   VAR
      ss_FB_HeartbeatPulse { ExternalAccessible := 'False'; ExternalVisible := 'False'; ExternalWritable := 'False'; S7_SetPoint := 'False'} : "FB_Pulse";   // Heartbeat send pulse generator
      s_UDT_MessageArray { ExternalAccessible := 'False'; ExternalVisible := 'False'; ExternalWritable := 'False'; S7_SetPoint := 'False'} : "UDT_MessageV2";   // Message array byte
      s_UDT_MessageHeader { ExternalAccessible := 'False'; ExternalVisible := 'False'; ExternalWritable := 'False'; S7_SetPoint := 'False'} : "UDT_MessageHeaderV2";   // Message header
      ss_Status { ExternalAccessible := 'False'; ExternalVisible := 'False'; ExternalWritable := 'False'} : Struct   // Status structure
         FIFOStatus { ExternalAccessible := 'False'; ExternalVisible := 'False'; ExternalWritable := 'False'} : "UDT_FifoStatus";
         FIFOError { ExternalAccessible := 'False'; ExternalVisible := 'False'; ExternalWritable := 'False'; S7_SetPoint := 'True'} : Bool;   //  FIFO error
         FIFOWarning { ExternalAccessible := 'False'; ExternalVisible := 'False'; ExternalWritable := 'False'; S7_SetPoint := 'True'} : Bool;   // FIFO warning
         InvalidMessageArraySize { ExternalAccessible := 'False'; ExternalVisible := 'False'; ExternalWritable := 'False'} : Bool;   // Message array is too short for message
         InvalidTimeInterval { ExternalAccessible := 'False'; ExternalVisible := 'False'; ExternalWritable := 'False'} : Bool;   // Heartbeat time interval lower than zero
      END_STRUCT;
      sdi_SerializePosition { ExternalAccessible := 'False'; ExternalVisible := 'False'; ExternalWritable := 'False'} : DInt;   // Position in array where serialize finished writing data +1
      si_MaximumMessageLength { ExternalAccessible := 'False'; ExternalVisible := 'False'; ExternalWritable := 'False'} : Int;   // Maximum number of elements in message array
      si_SerializeStatus { ExternalAccessible := 'False'; ExternalVisible := 'False'; ExternalWritable := 'False'} : Int;   // Function serialize status
      sx_HeartbeatPulse { ExternalAccessible := 'False'; ExternalVisible := 'False'; ExternalWritable := 'False'} : Bool;   // Heartbeat pulse
   END_VAR

   VAR CONSTANT
      ci_MessageID : Int := 20;   // Message ID number
      ci_MessageLength : Int := 18;   // Message length in bytes
   END_VAR


BEGIN
	(*
	----------------------------------------------------------------------------------------
	|                                                                                      |
	|  Copyright  2023             FORTNA Europe BV                                        |
	|  All Rights Reserved         Netherlands                                             |
	|                                                                                      |
	----------------------------------------------------------------------------------------
	Version history:
	Date        | Version   | Author       | Remark
	----------------------------------------------------------------------------------------
	03/01/2023  | 1.0       | S. Nikodem   | Release TIA 17 | DHL Munich 2023
	13/03/2023  | 1.1       | S. Nieswiec  | Updated for new Baseline
	*)
	REGION 1 – FIFO header status update

	    // Mode 'S' - FIFO register status update.
	    "FC_Fifo"(ic_Mode := 'S',
	              qUDT_Status => #ss_Status.FIFOStatus,
	              qx_Error => #ss_Status.FIFOError,
	              qx_Warning => #ss_Status.FIFOWarning,
	              iqv_Data := #s_UDT_MessageArray,
	              iqUDT_FifoHeader := #iq_UDT_FifoHeader,
	              iqv_DataBuffer := #iqs_FifoData);

	END_REGION

	REGION 2 – Heartbeat interval validation

	    // Check Heartbeat interval.
	    #ss_Status.InvalidTimeInterval := #iudi_HeartbeatInterval <= 0;

	END_REGION

	REGION 3 – Message array size validation

	    // Get size of the array.
	    #si_MaximumMessageLength := "FC_GetNrOfArrayEl"(#s_UDT_MessageArray.Bytes);

	    // Message array size validation.
	    #ss_Status.InvalidMessageArraySize := #ci_MessageLength > #si_MaximumMessageLength;

	END_REGION

	REGION 4 - Generate heartbeat pulse

	    IF NOT #ss_Status.InvalidTimeInterval
	        AND NOT #ss_Status.InvalidMessageArraySize
	    THEN
	        // Heartbeat pulse generator.
	        #ss_FB_HeartbeatPulse(iudi_PulseTime := #iudi_HeartbeatInterval,
	                              qx_Pulse => #sx_HeartbeatPulse);
	    END_IF;

	END_REGION

	REGION 5 – Message preparation

	    // FIFO full check.
	    IF NOT #iq_UDT_FifoHeader.Status.Full
	    THEN
	        // Errors and send pulse check.
	        IF NOT #ss_Status.FIFOError
	            AND NOT #ss_Status.InvalidMessageArraySize
	            AND #sx_HeartbeatPulse
	        THEN

	            REGION 5.1 – Header preparation

	                // Check sequence number. If it is equal or greater than 30000 reset it to 1.
	                IF #iqdi_MessageSequenceNumber < 30000
	                THEN
	                    #iqdi_MessageSequenceNumber += 1;
	                ELSE
	                    #iqdi_MessageSequenceNumber := 1;
	                END_IF;

	                // Write parts of the header into structure.
	                #s_UDT_MessageHeader.BodyLength := 0;
	                #s_UDT_MessageHeader.FlagRetry.%X0 := #ix_FlagRetry;
	                #s_UDT_MessageHeader.Group := #ii_MessageGroup;
	                #s_UDT_MessageHeader.MessageID := #ci_MessageID;
	                #s_UDT_MessageHeader.SequenceNumber := #iqdi_MessageSequenceNumber;
	                #s_UDT_MessageHeader.TimeSpan := #idi_TimeSpan;

	                // Calculate the header checksum.
	                "FC_Checksum"(i_UDT_MessageHeader := #s_UDT_MessageHeader,
	                              qb_Checksum => #s_UDT_MessageHeader.Checksum);

	            END_REGION

	            REGION 5.2 – Convert header into array of bytes

	                // Initialize the header serialize position and convert header structure into array of bytes.
	                #sdi_SerializePosition := 0;
	                #si_SerializeStatus := Serialize(SRC_VARIABLE := #s_UDT_MessageHeader,
	                                                 DEST_ARRAY => #s_UDT_MessageArray.Bytes,
	                                                 POS := #sdi_SerializePosition);

	            END_REGION

	            REGION 5.3 – Write message into the FIFO buffer

	                // Mode 'W' - Write FIFO record.
	                "FC_Fifo"(ic_Mode := 'W',
	                          qUDT_Status => #ss_Status.FIFOStatus,
	                          qx_Error => #ss_Status.FIFOError,
	                          qx_Warning => #ss_Status.FIFOWarning,
	                          iqv_Data := #s_UDT_MessageArray,
	                          iqUDT_FifoHeader := #iq_UDT_FifoHeader,
	                          iqv_DataBuffer := #iqs_FifoData);

	            END_REGION

	        END_IF;
	    ELSE
	        // If FIFO is full set FIFO main and FIFO full errors.
	        #ss_Status.FIFOError := TRUE;
	        #ss_Status.FIFOStatus.FifoFull := TRUE;
	    END_IF;

	END_REGION

	REGION 6 - Status

	    // Parametrization collective error output.
	    #qx_Error :=
	    #ss_Status.FIFOError
	    OR #ss_Status.InvalidTimeInterval
	    OR #ss_Status.InvalidMessageArraySize;

	    // Parametrization collective warning output.
	    #qx_Warning := #ss_Status.FIFOWarning;

	END_REGION
END_FUNCTION_BLOCK

FUNCTION_BLOCK "FB_MFC_Visu_PNNode_Status"
{ S7_Optimized_Access := 'TRUE' }
VERSION : 0.1
// ATTRIBUTES
// AUTO_NUMBER = True
// BLOCK_NUMBER = 155
// END_ATTRIBUTES
   VAR_INPUT
      i_UDT_PNNodeStatus { ExternalAccessible := 'False'; ExternalVisible := 'False'; ExternalWritable := 'False'} : "UDT_PNNodeStatus";   // PNNode status structure
      i_UDT_EquipmentNumber { ExternalAccessible := 'False'; ExternalVisible := 'False'; ExternalWritable := 'False'} : "UDT_EquipmentNumber";   // Item number
      ix_SendAllErrorsState { ExternalAccessible := 'False'; ExternalVisible := 'False'; ExternalWritable := 'False'} : Bool;   // True - update all the messages
      ix_MFCConnected { ExternalAccessible := 'False'; ExternalVisible := 'False'; ExternalWritable := 'False'} : Bool;   // True - A connection to the MFC has been established
      ix_CollectiveReset { ExternalAccessible := 'False'; ExternalVisible := 'False'; ExternalWritable := 'False'} : Bool;   // True - Collective reset command of all system controls
   END_VAR

   VAR_OUTPUT
      qx_Error { ExternalAccessible := 'False'; ExternalVisible := 'False'; ExternalWritable := 'False'} : Bool;   // Block error
      qx_Warning { ExternalAccessible := 'False'; ExternalVisible := 'False'; ExternalWritable := 'False'} : Bool;   // Block warning
   END_VAR

   VAR_IN_OUT
      iq_UDT_FifoHeader : "UDT_FifoHeader";   // FIFO header
      iqs_FifoData : Array[*] of "UDT_MessageV2";   // FIFO data buffer
      iqdi_MessageSequenceNumber { ExternalAccessible := 'False'; ExternalVisible := 'False'; ExternalWritable := 'False'} : DInt;   // Message number
   END_VAR

   VAR
      s_FB_ItemError { ExternalAccessible := 'False'; ExternalVisible := 'False'; ExternalWritable := 'False'; S7_SetPoint := 'False'} : "FB_ItemError";   // Item error block's instance
      s_FB_ItemStatus { ExternalAccessible := 'False'; ExternalVisible := 'False'; ExternalWritable := 'False'; S7_SetPoint := 'False'} : "FB_ItemStatus";   // Item status block's instance
      ss_FIFOStatus { ExternalAccessible := 'False'; ExternalVisible := 'False'; ExternalWritable := 'False'; S7_SetPoint := 'False'} : "UDT_FifoStatus";   // Status structure
      s_UDT_Message { ExternalAccessible := 'False'; ExternalVisible := 'False'; ExternalWritable := 'False'; S7_SetPoint := 'False'} : "UDT_MessageV2";   // Message
      s_UDT_PNNodeOld { ExternalAccessible := 'False'; ExternalVisible := 'False'; ExternalWritable := 'False'; S7_SetPoint := 'False'} : "UDT_PNNodeStatus";   // PNNode old status structure
      s_UDT_ItemError { ExternalAccessible := 'False'; ExternalVisible := 'False'; ExternalWritable := 'False'; S7_SetPoint := 'False'} : "UDT_ItemError";   // Item error message body structure
      s_UDT_ItemStatus { ExternalAccessible := 'False'; ExternalVisible := 'False'; ExternalWritable := 'False'; S7_SetPoint := 'False'} : "UDT_ItemStatus";   // Item status message body structure
      s_R_TRIG_Connection {InstructionName := 'R_TRIG'; LibVersion := '1.0'; ExternalAccessible := 'False'; ExternalVisible := 'False'; ExternalWritable := 'False'; S7_SetPoint := 'False'} : R_TRIG;   // Rising edge trigger connection reastablished
      s_F_TRIG_SendAllErrors {InstructionName := 'F_TRIG'; LibVersion := '1.0'; ExternalAccessible := 'False'; ExternalVisible := 'False'; ExternalWritable := 'False'; S7_SetPoint := 'False'} : F_TRIG;   // Falling edge trigger from signal send all errors
      sdi_Code { ExternalAccessible := 'False'; ExternalVisible := 'False'; ExternalWritable := 'False'} : DInt;   // Error code
      si_ItemStatus { ExternalAccessible := 'False'; ExternalVisible := 'False'; ExternalWritable := 'False'} : Int;   // Item status
      ii_ErrorNumber { ExternalAccessible := 'False'; ExternalVisible := 'False'; ExternalWritable := 'False'} : Int;   // Counter Error Number
      si_State { ExternalAccessible := 'False'; ExternalVisible := 'False'; ExternalWritable := 'False'} : Int;   // Error state
      sx_ItemErrorMessageReq { ExternalAccessible := 'False'; ExternalVisible := 'False'; ExternalWritable := 'False'} : Bool;   // Item error message required
      sx_ItemStatusMessageReq { ExternalAccessible := 'False'; ExternalVisible := 'False'; ExternalWritable := 'False'} : Bool;   // Item status message required
      sx_SendAllProcedure { ExternalAccessible := 'False'; ExternalVisible := 'False'; ExternalWritable := 'False'} : Bool;   // Send all procedure
      sx_FIFOError { ExternalAccessible := 'False'; ExternalVisible := 'False'; ExternalWritable := 'False'} : Bool;   // FIFO error
      sx_FIFOWarning { ExternalAccessible := 'False'; ExternalVisible := 'False'; ExternalWritable := 'False'} : Bool;   // FIFO warning
      sx_ItemErrorBlockError { ExternalAccessible := 'False'; ExternalVisible := 'False'; ExternalWritable := 'False'} : Bool;   // Item error block error
      sx_ItemErrorBlockWarning { ExternalAccessible := 'False'; ExternalVisible := 'False'; ExternalWritable := 'False'} : Bool;   // Item error block warning
      sx_ItemStatusBlockError { ExternalAccessible := 'False'; ExternalVisible := 'False'; ExternalWritable := 'False'} : Bool;   // Item status block error
      sx_ItemStatusBlockWarning { ExternalAccessible := 'False'; ExternalVisible := 'False'; ExternalWritable := 'False'} : Bool;   // Item status block warning
   END_VAR


BEGIN
	(*
	----------------------------------------------------------------------------------------
	|                                                                                      |
	|  Copyright  2023             FORTNA Europe BV                                        |
	|  All Rights Reserved         Netherlands                                             |
	|                                                                                      |
	----------------------------------------------------------------------------------------
	Version history:
	Date        | Version   | Author       | Remark
	----------------------------------------------------------------------------------------
	24/03/2023  | 1.0       | M. Diebel   | Release TIA 17 | DHL Munich 2023
	13/03/2023  | 1.1       | S. Nieswiec  | Updated for new Baseline
	*)


	REGION 1 - Initialize message required signals

	    #sx_ItemErrorMessageReq := FALSE;
	    #sx_ItemStatusMessageReq := FALSE;

	    // On connection reestablish send last remembered status and error state ( status only when it's diffrent then 0 )
	    #s_R_TRIG_Connection(CLK := #ix_MFCConnected);

	    IF #s_R_TRIG_Connection.Q AND #si_ItemStatus <> 0
	    THEN
	        #sx_ItemStatusMessageReq := TRUE;
	    END_IF;

	    IF #s_R_TRIG_Connection.Q
	    THEN
	        #sx_ItemErrorMessageReq := TRUE;
	    END_IF;

	    // Prepare trigger on the collective reset signal.
	    #s_F_TRIG_SendAllErrors(CLK := #ix_SendAllErrorsState);

	    // When collective reset will go down, start send every equipment errors.
	    IF #s_F_TRIG_SendAllErrors.Q AND NOT #sx_SendAllProcedure
	    THEN
	        #ii_ErrorNumber := 0;
	        #sx_SendAllProcedure := TRUE;
	    END_IF;

	END_REGION

	REGION 2 - FIFO header status update

	    // Mode 'S' - FIFO register status update.
	    "FC_Fifo"(ic_Mode := 'S',
	              qUDT_Status => #ss_FIFOStatus,
	              qx_Error => #sx_FIFOError,
	              qx_Warning => #sx_FIFOWarning,
	              iqv_Data := #s_UDT_Message,
	              iqUDT_FifoHeader := #iq_UDT_FifoHeader,
	              iqv_DataBuffer := #iqs_FifoData);

	END_REGION

	REGION 3 - Prepare message data

	    // When there is no reset errors command, update status and errors.
	    IF NOT #ix_CollectiveReset
	        AND NOT #ss_FIFOStatus.FifoPreFull
	    THEN
	        // Status
	        IF (#i_UDT_PNNodeStatus.Status <> #s_UDT_PNNodeOld.Status OR (#sx_SendAllProcedure AND #ii_ErrorNumber = 0))
	        THEN
	            #sx_ItemStatusMessageReq := TRUE;
	            #si_ItemStatus := #i_UDT_PNNodeStatus.Status;
	            #s_UDT_PNNodeOld.Status := #i_UDT_PNNodeStatus.Status;
	        END_IF;


	        // Check which specific status changed, prepare code, change state and write new status into the old one.
	        IF (#i_UDT_PNNodeStatus.Specific.PNSlaveNotOnline <> #s_UDT_PNNodeOld.Specific.PNSlaveNotOnline AND NOT #sx_SendAllProcedure)
	            OR (#sx_SendAllProcedure AND #ii_ErrorNumber = 0)
	        THEN
	            #sdi_Code := "DB_MFC_ErrorCode".PNNode.PNSlaveNotOnline;
	            #si_State := BOOL_TO_INT(#i_UDT_PNNodeStatus.Specific.PNSlaveNotOnline);
	            #s_UDT_PNNodeOld.Specific.PNSlaveNotOnline := #i_UDT_PNNodeStatus.Specific.PNSlaveNotOnline;
	            #sx_ItemErrorMessageReq := TRUE;
	            #ii_ErrorNumber += 1;
	        ELSIF (#i_UDT_PNNodeStatus.Specific.PNSlaveError <> #s_UDT_PNNodeOld.Specific.PNSlaveError AND NOT #sx_SendAllProcedure)
	            OR (#sx_SendAllProcedure AND #ii_ErrorNumber = 1)
	        THEN
	            #sdi_Code := "DB_MFC_ErrorCode".PNNode.PNSlaveError;
	            #si_State := BOOL_TO_INT(#i_UDT_PNNodeStatus.Specific.PNSlaveError);
	            #s_UDT_PNNodeOld.Specific.PNSlaveError := #i_UDT_PNNodeStatus.Specific.PNSlaveError;
	            #sx_ItemErrorMessageReq := TRUE;
	            #ii_ErrorNumber += 1;
	        ELSIF (#i_UDT_PNNodeStatus.Specific.PNSlaveWarning <> #s_UDT_PNNodeOld.Specific.PNSlaveWarning AND NOT #sx_SendAllProcedure)
	            OR (#sx_SendAllProcedure AND #ii_ErrorNumber = 2)
	        THEN
	            #sdi_Code := "DB_MFC_ErrorCode".PNNode.PNSlaveWarning;
	            #si_State := BOOL_TO_INT(#i_UDT_PNNodeStatus.Specific.PNSlaveWarning);
	            #s_UDT_PNNodeOld.Specific.PNSlaveWarning := #i_UDT_PNNodeStatus.Specific.PNSlaveWarning;
	            #sx_ItemErrorMessageReq := TRUE;
	            #sx_SendAllProcedure := FALSE;
	            #ii_ErrorNumber += 1;
	        END_IF;
	    END_IF;
	END_REGION

	REGION 4 - Write message components to the item error structure

	    #s_UDT_ItemError.ItemNumber := #i_UDT_EquipmentNumber;
	    #s_UDT_ItemError.Error := #sdi_Code;
	    #s_UDT_ItemError.State := #si_State;
	    #s_UDT_ItemError.Masked := 1;

	END_REGION

	REGION 5 - Write message components to the item status structure

	    #s_UDT_ItemStatus.Group := #i_UDT_EquipmentNumber.Group;
	    #s_UDT_ItemStatus.Node := #i_UDT_EquipmentNumber.Node;
	    #s_UDT_ItemStatus.Status := #si_ItemStatus;

	END_REGION

	REGION 6 - Prepare messages to the MFC

	    // If item error message required signal is set, prepare the item error message.
	    IF (#sx_ItemErrorMessageReq)
	    THEN
	        #s_FB_ItemError(i_UDT_ItemErrorBody := #s_UDT_ItemError,
	                        ii_MessageGroup := 1,
	                        ix_FlagRetry := FALSE,
	                        idi_TimeSpan := 0,
	                        qx_Error => #sx_ItemErrorBlockError,
	                        qx_Warning => #sx_ItemErrorBlockWarning,
	                        iq_UDT_FifoHeader := #iq_UDT_FifoHeader,
	                        iqs_FifoData := #iqs_FifoData,
	                        iqdi_MessageSequenceNumber := #iqdi_MessageSequenceNumber);
	    END_IF;

	    // If item status message required signal is set, prepare the item error message.
	    IF (#sx_ItemStatusMessageReq)
	    THEN
	        #s_FB_ItemStatus(i_UDT_ItemStatusBody := #s_UDT_ItemStatus,
	                         ii_MessageGroup := 1,
	                         ix_FlagRetry := FALSE,
	                         idi_TimeSpan := 0,
	                         qx_Error => #sx_ItemStatusBlockError,
	                         qx_Warning => #sx_ItemStatusBlockWarning,
	                         iq_UDT_FifoHeader := #iq_UDT_FifoHeader,
	                         iqs_FifoData := #iqs_FifoData,
	                         iqdi_MessageSequenceNumber := #iqdi_MessageSequenceNumber);
	    END_IF;

	END_REGION

	REGION 7 - Write outputs

	    // Prepare collective output error.
	    #qx_Error :=
	    #sx_ItemErrorBlockError
	    OR #sx_ItemStatusBlockError
	    OR #sx_FIFOError;

	    // Prepare collective output warning.
	    #qx_Warning :=
	    #sx_ItemErrorBlockWarning
	    OR #sx_ItemStatusBlockWarning
	    OR #sx_FIFOWarning;

	END_REGION
END_FUNCTION_BLOCK

FUNCTION_BLOCK "FB_MFC_Visu_EuchnerLock"
{ S7_Optimized_Access := 'TRUE' }
VERSION : 0.1
// ATTRIBUTES
// AUTO_NUMBER = True
// BLOCK_NUMBER = 149
// END_ATTRIBUTES
   VAR_INPUT
      i_UDT_EuchnerLock { ExternalAccessible := 'False'; ExternalVisible := 'False'; ExternalWritable := 'False'} : "UDT_EuchnerLockStatusV2";
      i_UDT_EquipmentNumber { ExternalAccessible := 'False'; ExternalVisible := 'False'; ExternalWritable := 'False'} : "UDT_EquipmentNumber";   // Item number
      ix_SendAllErrorsState { ExternalAccessible := 'False'; ExternalVisible := 'False'; ExternalWritable := 'False'} : Bool;   // True - update all the messages
      ix_MFCConnected { ExternalAccessible := 'False'; ExternalVisible := 'False'; ExternalWritable := 'False'} : Bool;   // True - A connection to the MFC has been established
      ix_CollectiveReset { ExternalAccessible := 'False'; ExternalVisible := 'False'; ExternalWritable := 'False'} : Bool;   // True - Collective reset command of all system controls
   END_VAR

   VAR_OUTPUT
      qx_Error { ExternalAccessible := 'False'; ExternalVisible := 'False'; ExternalWritable := 'False'} : Bool;   // Block error
      qx_Warning { ExternalAccessible := 'False'; ExternalVisible := 'False'; ExternalWritable := 'False'} : Bool;   // Block warning
   END_VAR

   VAR_IN_OUT
      iq_UDT_FifoHeader : "UDT_FifoHeader";   // FIFO header
      iqs_FifoData : Array[*] of "UDT_MessageV2";   // FIFO data buffer
      iqdi_MessageSequenceNumber { ExternalAccessible := 'False'; ExternalVisible := 'False'; ExternalWritable := 'False'} : DInt;   // Message number
   END_VAR

   VAR
      s_FB_ItemError { ExternalAccessible := 'False'; ExternalVisible := 'False'; ExternalWritable := 'False'; S7_SetPoint := 'False'} : "FB_ItemError";   // Item error block's instance
      s_FB_ItemStatus { ExternalAccessible := 'False'; ExternalVisible := 'False'; ExternalWritable := 'False'; S7_SetPoint := 'False'} : "FB_ItemStatus";   // Item status block's instance
      ss_FIFOStatus { ExternalAccessible := 'False'; ExternalVisible := 'False'; ExternalWritable := 'False'; S7_SetPoint := 'False'} : "UDT_FifoStatus";   // Status structure
      s_UDT_Message { ExternalAccessible := 'False'; ExternalVisible := 'False'; ExternalWritable := 'False'; S7_SetPoint := 'False'} : "UDT_MessageV2";   // Message
      s_UDT_EuchnerLockOld { ExternalAccessible := 'False'; ExternalVisible := 'False'; ExternalWritable := 'False'; S7_SetPoint := 'False'} : "UDT_EuchnerLockStatusV2";   // ColumnLift status structure
      s_UDT_ItemError { ExternalAccessible := 'False'; ExternalVisible := 'False'; ExternalWritable := 'False'; S7_SetPoint := 'False'} : "UDT_ItemError";   // Item error message body structure
      s_UDT_ItemStatus { ExternalAccessible := 'False'; ExternalVisible := 'False'; ExternalWritable := 'False'; S7_SetPoint := 'False'} : "UDT_ItemStatus";   // Item status message body structure
      s_R_TRIG_Connection {InstructionName := 'R_TRIG'; LibVersion := '1.0'; ExternalAccessible := 'False'; ExternalVisible := 'False'; ExternalWritable := 'False'; S7_SetPoint := 'False'} : R_TRIG;   // Rising edge trigger connection reastablished
      s_F_TRIG_SendAllErrors {InstructionName := 'F_TRIG'; LibVersion := '1.0'; ExternalAccessible := 'False'; ExternalVisible := 'False'; ExternalWritable := 'False'; S7_SetPoint := 'False'} : F_TRIG;   // Falling edge trigger from signal send all errors
      sdi_Code { ExternalAccessible := 'False'; ExternalVisible := 'False'; ExternalWritable := 'False'} : DInt;   // Error code
      si_ItemStatus { ExternalAccessible := 'False'; ExternalVisible := 'False'; ExternalWritable := 'False'} : Int;   // Item status
      ii_ErrorNumber { ExternalAccessible := 'False'; ExternalVisible := 'False'; ExternalWritable := 'False'} : Int;   // Counter Error Number
      si_State { ExternalAccessible := 'False'; ExternalVisible := 'False'; ExternalWritable := 'False'} : Int;   // Error state
      sx_ItemErrorMessageReq { ExternalAccessible := 'False'; ExternalVisible := 'False'; ExternalWritable := 'False'} : Bool;   // Item error message required
      sx_ItemStatusMessageReq { ExternalAccessible := 'False'; ExternalVisible := 'False'; ExternalWritable := 'False'} : Bool;   // Item status message required
      sx_SendAllProcedure { ExternalAccessible := 'False'; ExternalVisible := 'False'; ExternalWritable := 'False'} : Bool;   // Send all procedure
      sx_FIFOError { ExternalAccessible := 'False'; ExternalVisible := 'False'; ExternalWritable := 'False'} : Bool;   // FIFO error
      sx_FIFOWarning { ExternalAccessible := 'False'; ExternalVisible := 'False'; ExternalWritable := 'False'} : Bool;   // FIFO warning
      sx_ItemErrorBlockError { ExternalAccessible := 'False'; ExternalVisible := 'False'; ExternalWritable := 'False'} : Bool;   // Item error block error
      sx_ItemErrorBlockWarning { ExternalAccessible := 'False'; ExternalVisible := 'False'; ExternalWritable := 'False'} : Bool;   // Item error block warning
      sx_ItemStatusBlockError { ExternalAccessible := 'False'; ExternalVisible := 'False'; ExternalWritable := 'False'} : Bool;   // Item status block error
      sx_ItemStatusBlockWarning { ExternalAccessible := 'False'; ExternalVisible := 'False'; ExternalWritable := 'False'} : Bool;   // Item status block warning
      s_UDT_EuchnerLockStatus { ExternalAccessible := 'False'; ExternalVisible := 'False'; ExternalWritable := 'False'; S7_SetPoint := 'False'} : "UDT_EuchnerLockStatusV2";   // ColumnLift status structure
   END_VAR


BEGIN
	(*
	----------------------------------------------------------------------------------------
	|                                                                                      |
	|  Copyright  2023             FORTNA Europe BV                                        |
	|  All Rights Reserved         Netherlands                                             |
	|                                                                                      |
	----------------------------------------------------------------------------------------
	Version history:
	Date        | Version   | Author       | Remark
	----------------------------------------------------------------------------------------
	10/10/2023  | 1.0       | M. Diebel   | Release TIA 17 | DHL Munich 2023
	06/02/2024  | 1.1       | L.Klar      | New alarms added
	13/03/2023  | 1.2       | S. Nieswiec  | Updated for new Baseline
	*)


	REGION 1 - Initialize message required signals


	    #sx_ItemErrorMessageReq := FALSE;
	    #sx_ItemStatusMessageReq := FALSE;

	    // On connection reestablish send last remembered status and error state ( status only when it's diffrent then 0 )
	    #s_R_TRIG_Connection(CLK := #ix_MFCConnected);

	    IF #s_R_TRIG_Connection.Q AND #si_ItemStatus <> 0
	    THEN
	        #sx_ItemStatusMessageReq := TRUE;
	    END_IF;

	    IF #s_R_TRIG_Connection.Q
	    THEN
	        #sx_ItemErrorMessageReq := TRUE;
	    END_IF;

	    // Prepare trigger on the collective reset signal.
	    #s_F_TRIG_SendAllErrors(CLK := #ix_SendAllErrorsState);

	    // When collective reset will go down, start send every equipment errors.
	    IF #s_F_TRIG_SendAllErrors.Q AND NOT #sx_SendAllProcedure
	    THEN
	        #ii_ErrorNumber := 0;
	        #sx_SendAllProcedure := TRUE;
	    END_IF;

	END_REGION

	REGION 2 - FIFO header status update

	    // Mode 'S' - FIFO register status update.
	    "FC_Fifo"(ic_Mode := 'S',
	              qUDT_Status => #ss_FIFOStatus,
	              qx_Error => #sx_FIFOError,
	              qx_Warning => #sx_FIFOWarning,
	              iqv_Data := #s_UDT_Message,
	              iqUDT_FifoHeader := #iq_UDT_FifoHeader,
	              iqv_DataBuffer := #iqs_FifoData);

	END_REGION

	REGION 3 - Prepare message data

	    //
	    #s_UDT_EuchnerLockStatus := #i_UDT_EuchnerLock;
	    // When there is no reset errors command, update status and errors.
	    IF NOT #ix_CollectiveReset
	        AND NOT #ss_FIFOStatus.FifoPreFull
	    THEN


	        // Check which specific status changed, prepare code, change state and write new status into the old one.
	        IF (#s_UDT_EuchnerLockStatus.LockFault <> #s_UDT_EuchnerLockOld.LockFault AND NOT #sx_SendAllProcedure)
	            OR (#sx_SendAllProcedure AND #ii_ErrorNumber = 0)
	        THEN
	            #sdi_Code := "DB_MFC_ErrorCode".EuchnerLock.LockFault;
	            #si_State := BOOL_TO_INT(#s_UDT_EuchnerLockStatus.LockFault);
	            #s_UDT_EuchnerLockOld.LockFault := #s_UDT_EuchnerLockStatus.LockFault;
	            #sx_ItemErrorMessageReq := TRUE;
	            #ii_ErrorNumber += 1;
	        ELSIF (#s_UDT_EuchnerLockStatus.DoorClosed <> #s_UDT_EuchnerLockOld.DoorClosed AND NOT #sx_SendAllProcedure)
	            OR (#sx_SendAllProcedure AND #ii_ErrorNumber = 1)
	        THEN
	            #sdi_Code := "DB_MFC_ErrorCode".EuchnerLock.DoorClosed;
	            #si_State := BOOL_TO_INT(#s_UDT_EuchnerLockStatus.DoorClosed);
	            #s_UDT_EuchnerLockOld.DoorClosed := #s_UDT_EuchnerLockStatus.DoorClosed;
	            #sx_ItemErrorMessageReq := TRUE;
	            #ii_ErrorNumber += 1;
	        ELSIF (#s_UDT_EuchnerLockStatus.DoorOpened <> #s_UDT_EuchnerLockOld.DoorOpened AND NOT #sx_SendAllProcedure)
	            OR (#sx_SendAllProcedure AND #ii_ErrorNumber = 2)
	        THEN
	            #sdi_Code := "DB_MFC_ErrorCode".EuchnerLock.DoorOpened;
	            #si_State := BOOL_TO_INT(#s_UDT_EuchnerLockStatus.DoorOpened);
	            #s_UDT_EuchnerLockOld.DoorOpened := #s_UDT_EuchnerLockStatus.DoorOpened;
	            #sx_ItemErrorMessageReq := TRUE;
	            #ii_ErrorNumber += 1;
	        ELSIF (#s_UDT_EuchnerLockStatus.BoltTongueClosed <> #s_UDT_EuchnerLockOld.BoltTongueClosed AND NOT #sx_SendAllProcedure)
	            OR (#sx_SendAllProcedure AND #ii_ErrorNumber = 3)
	        THEN
	            #sdi_Code := "DB_MFC_ErrorCode".EuchnerLock.BoltTongueClosed;
	            #si_State := BOOL_TO_INT(#s_UDT_EuchnerLockStatus.BoltTongueClosed);
	            #s_UDT_EuchnerLockOld.BoltTongueClosed := #s_UDT_EuchnerLockStatus.BoltTongueClosed;
	            #sx_ItemErrorMessageReq := TRUE;
	            #ii_ErrorNumber += 1;
	        ELSIF (#s_UDT_EuchnerLockStatus.Safelylocked <> #s_UDT_EuchnerLockOld.Safelylocked AND NOT #sx_SendAllProcedure)
	            OR (#sx_SendAllProcedure AND #ii_ErrorNumber = 4)
	        THEN
	            #sdi_Code := "DB_MFC_ErrorCode".EuchnerLock.Safelylocked;
	            #si_State := BOOL_TO_INT(#s_UDT_EuchnerLockStatus.Safelylocked);
	            #s_UDT_EuchnerLockOld.Safelylocked := #s_UDT_EuchnerLockStatus.Safelylocked;
	            #sx_ItemErrorMessageReq := TRUE;
	            #ii_ErrorNumber += 1;
	        ELSIF (#s_UDT_EuchnerLockStatus.SafetyLockAckReq <> #s_UDT_EuchnerLockOld.SafetyLockAckReq AND NOT #sx_SendAllProcedure)
	            OR (#sx_SendAllProcedure AND #ii_ErrorNumber = 5)
	        THEN
	            #sdi_Code := "DB_MFC_ErrorCode".EuchnerLock.SafetyLockAckReq;
	            #si_State := BOOL_TO_INT(#s_UDT_EuchnerLockStatus.SafetyLockAckReq);
	            #s_UDT_EuchnerLockOld.SafetyLockAckReq := #s_UDT_EuchnerLockStatus.SafetyLockAckReq;
	            #sx_ItemErrorMessageReq := TRUE;
	            #ii_ErrorNumber += 1;
	        ELSIF (#s_UDT_EuchnerLockStatus.ReqMissingAccessRights <> #s_UDT_EuchnerLockOld.ReqMissingAccessRights AND NOT #sx_SendAllProcedure)
	            OR (#sx_SendAllProcedure AND #ii_ErrorNumber = 6)
	        THEN
	            #sdi_Code := "DB_MFC_ErrorCode".EuchnerLock.ReqMissingAccessRights;
	            #si_State := BOOL_TO_INT(#s_UDT_EuchnerLockStatus.ReqMissingAccessRights);
	            #s_UDT_EuchnerLockOld.ReqMissingAccessRights := #s_UDT_EuchnerLockStatus.ReqMissingAccessRights;
	            #sx_ItemErrorMessageReq := TRUE;
	            #ii_ErrorNumber += 1;
	        ELSIF (#s_UDT_EuchnerLockStatus.ResetMissingAccessRights <> #s_UDT_EuchnerLockOld.ResetMissingAccessRights AND NOT #sx_SendAllProcedure)
	            OR (#sx_SendAllProcedure AND #ii_ErrorNumber = 7)
	        THEN
	            #sdi_Code := "DB_MFC_ErrorCode".EuchnerLock.ResetMissingAccessRights;
	            #si_State := BOOL_TO_INT(#s_UDT_EuchnerLockStatus.ResetMissingAccessRights);
	            #s_UDT_EuchnerLockOld.ResetMissingAccessRights := #s_UDT_EuchnerLockStatus.ResetMissingAccessRights;
	            #sx_ItemErrorMessageReq := TRUE;
	            #ii_ErrorNumber += 1;
	        ELSIF (#s_UDT_EuchnerLockStatus.DoorOpenedWithoutReq <> #s_UDT_EuchnerLockOld.DoorOpenedWithoutReq AND NOT #sx_SendAllProcedure)
	            OR (#sx_SendAllProcedure AND #ii_ErrorNumber = 8)
	        THEN
	            #sdi_Code := "DB_MFC_ErrorCode".EuchnerLock.DoorOpenedWithoutReq;
	            #si_State := BOOL_TO_INT(#s_UDT_EuchnerLockStatus.DoorOpenedWithoutReq);
	            #s_UDT_EuchnerLockOld.DoorOpenedWithoutReq := #s_UDT_EuchnerLockStatus.DoorOpenedWithoutReq;
	            #sx_ItemErrorMessageReq := TRUE;
	            #ii_ErrorNumber += 1;
	            #sx_SendAllProcedure := FALSE;
	        END_IF;
	    END_IF;
	END_REGION

	REGION 4 - Write message components to the item error structure

	    #s_UDT_ItemError.ItemNumber := #i_UDT_EquipmentNumber;
	    #s_UDT_ItemError.Error := #sdi_Code;
	    #s_UDT_ItemError.State := #si_State;
	    #s_UDT_ItemError.Masked := 1;

	END_REGION

	REGION 5 - Write message components to the item status structure

	    #s_UDT_ItemStatus.Group := #i_UDT_EquipmentNumber.Group;
	    #s_UDT_ItemStatus.Node := #i_UDT_EquipmentNumber.Node;
	    #s_UDT_ItemStatus.Status := #si_ItemStatus;

	END_REGION

	REGION 6 - Prepare messages to the MFC

	    // If item error message required signal is set, prepare the item error message.
	    IF (#sx_ItemErrorMessageReq)
	    THEN
	        #s_FB_ItemError(i_UDT_ItemErrorBody := #s_UDT_ItemError,
	                        ii_MessageGroup := 1,
	                        ix_FlagRetry := FALSE,
	                        idi_TimeSpan := 0,
	                        qx_Error => #sx_ItemErrorBlockError,
	                        qx_Warning => #sx_ItemErrorBlockWarning,
	                        iq_UDT_FifoHeader := #iq_UDT_FifoHeader,
	                        iqs_FifoData := #iqs_FifoData,
	                        iqdi_MessageSequenceNumber := #iqdi_MessageSequenceNumber);
	    END_IF;

	    // If item status message required signal is set, prepare the item error message.
	    IF (#sx_ItemStatusMessageReq)
	    THEN
	        #s_FB_ItemStatus(i_UDT_ItemStatusBody := #s_UDT_ItemStatus,
	                         ii_MessageGroup := 1,
	                         ix_FlagRetry := FALSE,
	                         idi_TimeSpan := 0,
	                         qx_Error => #sx_ItemStatusBlockError,
	                         qx_Warning => #sx_ItemStatusBlockWarning,
	                         iq_UDT_FifoHeader := #iq_UDT_FifoHeader,
	                         iqs_FifoData := #iqs_FifoData,
	                         iqdi_MessageSequenceNumber := #iqdi_MessageSequenceNumber);
	    END_IF;

	END_REGION

	REGION 7 - Write outputs

	    // Prepare collective output error.
	    #qx_Error :=
	    #sx_ItemErrorBlockError
	    OR #sx_ItemStatusBlockError
	    OR #sx_FIFOError;

	    // Prepare collective output warning.
	    #qx_Warning :=
	    #sx_ItemErrorBlockWarning
	    OR #sx_ItemStatusBlockWarning
	    OR #sx_FIFOWarning;

	END_REGION
END_FUNCTION_BLOCK

FUNCTION_BLOCK "FB_MFC_Visu_EStop_Status"
{ S7_Optimized_Access := 'TRUE' }
VERSION : 0.1
// ATTRIBUTES
// AUTO_NUMBER = True
// BLOCK_NUMBER = 148
// END_ATTRIBUTES
   VAR_INPUT
      i_UDT_EStopStatus { ExternalAccessible := 'False'; ExternalVisible := 'False'; ExternalWritable := 'False'} : "UDT_EStop_Status";   // EStop status structure
      i_UDT_EquipmentNumber { ExternalAccessible := 'False'; ExternalVisible := 'False'; ExternalWritable := 'False'} : "UDT_EquipmentNumber";   // Item number
      ix_SendAllErrorsState { ExternalAccessible := 'False'; ExternalVisible := 'False'; ExternalWritable := 'False'} : Bool;   // True - update all the messages
      ix_MFCConnected { ExternalAccessible := 'False'; ExternalVisible := 'False'; ExternalWritable := 'False'} : Bool;   // True - A connection to the MFC has been established
      ix_CollectiveReset { ExternalAccessible := 'False'; ExternalVisible := 'False'; ExternalWritable := 'False'} : Bool;   // True - Collective reset command of all system controls
   END_VAR

   VAR_OUTPUT
      qx_Error { ExternalAccessible := 'False'; ExternalVisible := 'False'; ExternalWritable := 'False'} : Bool;   // Block error
      qx_Warning { ExternalAccessible := 'False'; ExternalVisible := 'False'; ExternalWritable := 'False'} : Bool;   // Block warning
   END_VAR

   VAR_IN_OUT
      iq_UDT_FifoHeader : "UDT_FifoHeader";   // FIFO header
      iqs_FifoData : Array[*] of "UDT_MessageV2";   // FIFO data buffer
      iqdi_MessageSequenceNumber { ExternalAccessible := 'False'; ExternalVisible := 'False'; ExternalWritable := 'False'} : DInt;   // Message number
   END_VAR

   VAR
      s_FB_ItemStatus { ExternalAccessible := 'False'; ExternalVisible := 'False'; ExternalWritable := 'False'; S7_SetPoint := 'False'} : "FB_ItemStatus";   // Item status block's instance
      s_FB_ItemError { ExternalAccessible := 'False'; ExternalVisible := 'False'; ExternalWritable := 'False'; S7_SetPoint := 'False'} : "FB_ItemError";   // Item error block's instance
      ss_FIFOStatus { ExternalAccessible := 'False'; ExternalVisible := 'False'; ExternalWritable := 'False'; S7_SetPoint := 'False'} : "UDT_FifoStatus";   // Status structure
      s_UDT_Message { ExternalAccessible := 'False'; ExternalVisible := 'False'; ExternalWritable := 'False'; S7_SetPoint := 'False'} : "UDT_MessageV2";   // Message
      s_UDT_EStopOld { ExternalAccessible := 'False'; ExternalVisible := 'False'; ExternalWritable := 'False'; S7_SetPoint := 'False'} : "UDT_EStop_Status";   // EStop  status structure
      s_UDT_ItemError { ExternalAccessible := 'False'; ExternalVisible := 'False'; ExternalWritable := 'False'; S7_SetPoint := 'False'} : "UDT_ItemError";   // Item error message body structure
      s_UDT_ItemStatus { ExternalAccessible := 'False'; ExternalVisible := 'False'; ExternalWritable := 'False'; S7_SetPoint := 'False'} : "UDT_ItemStatus";   // Item status message body structure
      s_F_TRIG_SendAllErrors {InstructionName := 'F_TRIG'; LibVersion := '1.0'; ExternalAccessible := 'False'; ExternalVisible := 'False'; ExternalWritable := 'False'; S7_SetPoint := 'False'} : F_TRIG;   // Falling edge trigger from signal send all errors
      s_R_TRIG_Connection {InstructionName := 'R_TRIG'; LibVersion := '1.0'; ExternalAccessible := 'False'; ExternalVisible := 'False'; ExternalWritable := 'False'; S7_SetPoint := 'False'} : R_TRIG;   // Rising edge trigger connection reastablished
      sdi_Code { ExternalAccessible := 'False'; ExternalVisible := 'False'; ExternalWritable := 'False'} : DInt;   // Error code
      si_ItemStatus { ExternalAccessible := 'False'; ExternalVisible := 'False'; ExternalWritable := 'False'} : Int;   // Item status
      ii_ErrorNumber { ExternalAccessible := 'False'; ExternalVisible := 'False'; ExternalWritable := 'False'} : Int;   // Counter Error Number
      si_State { ExternalAccessible := 'False'; ExternalVisible := 'False'; ExternalWritable := 'False'} : Int;   // Error state
      sx_ItemErrorMessageReq { ExternalAccessible := 'False'; ExternalVisible := 'False'; ExternalWritable := 'False'} : Bool;   // Item error message required
      sx_ItemStatusMessageReq { ExternalAccessible := 'False'; ExternalVisible := 'False'; ExternalWritable := 'False'} : Bool;   // Item status message required
      sx_SendAllProcedure { ExternalAccessible := 'False'; ExternalVisible := 'False'; ExternalWritable := 'False'} : Bool;   // Send all procedure
      sx_FIFOError { ExternalAccessible := 'False'; ExternalVisible := 'False'; ExternalWritable := 'False'} : Bool;   // FIFO error
      sx_FIFOWarning { ExternalAccessible := 'False'; ExternalVisible := 'False'; ExternalWritable := 'False'} : Bool;   // FIFO warning
      sx_ItemErrorBlockError { ExternalAccessible := 'False'; ExternalVisible := 'False'; ExternalWritable := 'False'} : Bool;   // Item error block error
      sx_ItemErrorBlockWarning { ExternalAccessible := 'False'; ExternalVisible := 'False'; ExternalWritable := 'False'} : Bool;   // Item error block warning
      sx_ItemStatusBlockError { ExternalAccessible := 'False'; ExternalVisible := 'False'; ExternalWritable := 'False'} : Bool;   // Item status block error
      sx_ItemStatusBlockWarning { ExternalAccessible := 'False'; ExternalVisible := 'False'; ExternalWritable := 'False'} : Bool;   // Item status block warning
   END_VAR


BEGIN
	(*
	----------------------------------------------------------------------------------------
	|                                                                                      |
	|  Copyright  2023             FORTNA Europe BV                                        |
	|  All Rights Reserved         Netherlands                                             |
	|                                                                                      |
	----------------------------------------------------------------------------------------
	Version history:
	Date        | Version   | Author       | Remark
	----------------------------------------------------------------------------------------
	21/03/2023  | 1.0       | M. Diebel   | Release TIA 17 | DHL Munich 2023
	13/03/2023  | 1.1       | S. Nieswiec  | Updated for new Baseline
	*)


	REGION 1 - Initialize message required signals

	    #sx_ItemErrorMessageReq := FALSE;
	    #sx_ItemStatusMessageReq := FALSE;

	    // On connection reestablish send last remembered status and error state ( status only when it's diffrent then 0 )
	    #s_R_TRIG_Connection(CLK := #ix_MFCConnected);

	    IF #s_R_TRIG_Connection.Q AND #si_ItemStatus <> 0
	    THEN
	        #sx_ItemStatusMessageReq := TRUE;
	    END_IF;

	    IF #s_R_TRIG_Connection.Q
	    THEN
	        #sx_ItemErrorMessageReq := TRUE;
	    END_IF;

	    // Prepare trigger on the collective reset signal.
	    #s_F_TRIG_SendAllErrors(CLK := #ix_SendAllErrorsState);

	    // When collective reset will go down, start send every equipment errors.
	    IF #s_F_TRIG_SendAllErrors.Q AND NOT #sx_SendAllProcedure
	    THEN
	        #sx_SendAllProcedure := TRUE;
	    END_IF;

	END_REGION

	REGION 2 - FIFO header status update

	    // Mode 'S' - FIFO register status update.
	    "FC_Fifo"(ic_Mode := 'S',
	              qUDT_Status => #ss_FIFOStatus,
	              qx_Error => #sx_FIFOError,
	              qx_Warning => #sx_FIFOWarning,
	              iqv_Data := #s_UDT_Message,
	              iqUDT_FifoHeader := #iq_UDT_FifoHeader,
	              iqv_DataBuffer := #iqs_FifoData);

	END_REGION

	REGION 3 - Prepare message data

	    // When there is no reset errors command, update status and errors.
	    IF NOT #ix_CollectiveReset
	        AND NOT #ss_FIFOStatus.FifoPreFull
	    THEN
	        // Status
	        IF (#i_UDT_EStopStatus.Status <> #s_UDT_EStopOld.Status OR (#sx_SendAllProcedure))
	        THEN
	            #sx_ItemStatusMessageReq := TRUE;
	            #si_ItemStatus := #i_UDT_EStopStatus.Status;
	            #s_UDT_EStopOld.Status := #i_UDT_EStopStatus.Status;
	        END_IF;


	        // Check which specific status changed, prepare code, change state and write new status into the old one.
	        IF (#i_UDT_EStopStatus.Estop <> #s_UDT_EStopOld.Estop AND NOT #sx_SendAllProcedure)
	            OR (#sx_SendAllProcedure)
	        THEN
	            #sdi_Code := "DB_MFC_ErrorCode".EStop.EStop;
	            #si_State := BOOL_TO_INT(#i_UDT_EStopStatus.Estop);
	            #s_UDT_EStopOld.Estop := #i_UDT_EStopStatus.Estop;
	            #sx_ItemErrorMessageReq := TRUE;
	            #sx_SendAllProcedure := FALSE;
	        END_IF;
	    END_IF;
	END_REGION

	REGION 4 - Write message components to the item error structure

	    #s_UDT_ItemError.ItemNumber := #i_UDT_EquipmentNumber;
	    #s_UDT_ItemError.Error := #sdi_Code;
	    #s_UDT_ItemError.State := #si_State;
	    #s_UDT_ItemError.Masked := 1;

	END_REGION

	REGION 5 - Write message components to the item status structure

	    #s_UDT_ItemStatus.Group := #i_UDT_EquipmentNumber.Group;
	    #s_UDT_ItemStatus.Node := #i_UDT_EquipmentNumber.Node;
	    #s_UDT_ItemStatus.Status := #si_ItemStatus;

	END_REGION

	REGION 6 - Prepare messages to the MFC

	    // If item error message required signal is set, prepare the item error message.
	    IF (#sx_ItemErrorMessageReq)
	    THEN
	        #s_FB_ItemError(i_UDT_ItemErrorBody := #s_UDT_ItemError,
	                        ii_MessageGroup := 1,
	                        ix_FlagRetry := FALSE,
	                        idi_TimeSpan := 0,
	                        qx_Error => #sx_ItemErrorBlockError,
	                        qx_Warning => #sx_ItemErrorBlockWarning,
	                        iq_UDT_FifoHeader := #iq_UDT_FifoHeader,
	                        iqs_FifoData := #iqs_FifoData,
	                        iqdi_MessageSequenceNumber := #iqdi_MessageSequenceNumber);
	    END_IF;

	    // If item status message required signal is set, prepare the item error message.
	    IF (#sx_ItemStatusMessageReq)
	    THEN
	        #s_FB_ItemStatus(i_UDT_ItemStatusBody := #s_UDT_ItemStatus,
	                         ii_MessageGroup := 1,
	                         ix_FlagRetry := FALSE,
	                         idi_TimeSpan := 0,
	                         qx_Error => #sx_ItemStatusBlockError,
	                         qx_Warning => #sx_ItemStatusBlockWarning,
	                         iq_UDT_FifoHeader := #iq_UDT_FifoHeader,
	                         iqs_FifoData := #iqs_FifoData,
	                         iqdi_MessageSequenceNumber := #iqdi_MessageSequenceNumber);
	    END_IF;

	END_REGION

	REGION 7 - Write outputs

	    // Prepare collective output error.
	    #qx_Error :=
	    #sx_ItemErrorBlockError
	    OR #sx_ItemStatusBlockError
	    OR #sx_FIFOError;

	    // Prepare collective output warning.
	    #qx_Warning :=
	    #sx_ItemErrorBlockWarning
	    OR #sx_ItemStatusBlockWarning
	    OR #sx_FIFOWarning;

	END_REGION
END_FUNCTION_BLOCK

FUNCTION_BLOCK "FB_MFC_Visu_CPG_Status"
{ S7_Optimized_Access := 'TRUE' }
VERSION : 0.1
// ATTRIBUTES
// AUTO_NUMBER = True
// BLOCK_NUMBER = 142
// END_ATTRIBUTES
   VAR_INPUT
      i_UDT_CPGStatus { ExternalAccessible := 'False'; ExternalVisible := 'False'; ExternalWritable := 'False'} : "UDT_ControlPowerGroupWORStatus";   // CPG status structure
      i_UDT_EquipmentNumber { ExternalAccessible := 'False'; ExternalVisible := 'False'; ExternalWritable := 'False'} : "UDT_EquipmentNumber";   // Item number
      ix_SendAllErrorsState { ExternalAccessible := 'False'; ExternalVisible := 'False'; ExternalWritable := 'False'} : Bool;   // True - update all the messages
      ix_MFCConnected { ExternalAccessible := 'False'; ExternalVisible := 'False'; ExternalWritable := 'False'} : Bool;   // True - A connection to the MFC has been established
      ix_CollectiveReset { ExternalAccessible := 'False'; ExternalVisible := 'False'; ExternalWritable := 'False'} : Bool;   // True - Collective reset command of all system controls
   END_VAR

   VAR_OUTPUT
      qx_Error { ExternalAccessible := 'False'; ExternalVisible := 'False'; ExternalWritable := 'False'} : Bool;   // Block error
      qx_Warning { ExternalAccessible := 'False'; ExternalVisible := 'False'; ExternalWritable := 'False'} : Bool;   // Block warning
   END_VAR

   VAR_IN_OUT
      iq_UDT_FifoHeader : "UDT_FifoHeader";   // FIFO header
      iqs_FifoData : Array[*] of "UDT_MessageV2";   // FIFO data buffer
      iqdi_MessageSequenceNumber { ExternalAccessible := 'False'; ExternalVisible := 'False'; ExternalWritable := 'False'} : DInt;   // Message number
   END_VAR

   VAR
      s_FB_ItemError { ExternalAccessible := 'False'; ExternalVisible := 'False'; ExternalWritable := 'False'; S7_SetPoint := 'False'} : "FB_ItemError";   // Item error block's instance
      s_FB_ItemStatus { ExternalAccessible := 'False'; ExternalVisible := 'False'; ExternalWritable := 'False'; S7_SetPoint := 'False'} : "FB_ItemStatus";   // Item status block's instance
      ss_FIFOStatus { ExternalAccessible := 'False'; ExternalVisible := 'False'; ExternalWritable := 'False'; S7_SetPoint := 'False'} : "UDT_FifoStatus";   // Status structure
      s_UDT_Message { ExternalAccessible := 'False'; ExternalVisible := 'False'; ExternalWritable := 'False'; S7_SetPoint := 'False'} : "UDT_MessageV2";   // Message
      s_UDT_CPGOld { ExternalAccessible := 'False'; ExternalVisible := 'False'; ExternalWritable := 'False'; S7_SetPoint := 'False'} : "UDT_ControlPowerGroupStatus";   // CPG status structure
      s_UDT_ItemError { ExternalAccessible := 'False'; ExternalVisible := 'False'; ExternalWritable := 'False'; S7_SetPoint := 'False'} : "UDT_ItemError";   // Item error message body structure
      s_UDT_ItemStatus { ExternalAccessible := 'False'; ExternalVisible := 'False'; ExternalWritable := 'False'; S7_SetPoint := 'False'} : "UDT_ItemStatus";   // Item status message body structure
      s_R_TRIG_Connection {InstructionName := 'R_TRIG'; LibVersion := '1.0'; ExternalAccessible := 'False'; ExternalVisible := 'False'; ExternalWritable := 'False'; S7_SetPoint := 'False'} : R_TRIG;   // Rising edge trigger connection reastablished
      s_F_TRIG_SendAllErrors {InstructionName := 'F_TRIG'; LibVersion := '1.0'; ExternalAccessible := 'False'; ExternalVisible := 'False'; ExternalWritable := 'False'; S7_SetPoint := 'False'} : F_TRIG;   // Falling edge trigger from signal send all errors
      sdi_Code { ExternalAccessible := 'False'; ExternalVisible := 'False'; ExternalWritable := 'False'} : DInt;   // Error code
      si_ItemStatus { ExternalAccessible := 'False'; ExternalVisible := 'False'; ExternalWritable := 'False'} : Int;   // Item status
      ii_ErrorNumber { ExternalAccessible := 'False'; ExternalVisible := 'False'; ExternalWritable := 'False'} : Int;   // Counter Error Number
      si_State { ExternalAccessible := 'False'; ExternalVisible := 'False'; ExternalWritable := 'False'} : Int;   // Error state
      sx_ItemErrorMessageReq { ExternalAccessible := 'False'; ExternalVisible := 'False'; ExternalWritable := 'False'} : Bool;   // Item error message required
      sx_ItemStatusMessageReq { ExternalAccessible := 'False'; ExternalVisible := 'False'; ExternalWritable := 'False'} : Bool;   // Item status message required
      sx_SendAllProcedure { ExternalAccessible := 'False'; ExternalVisible := 'False'; ExternalWritable := 'False'} : Bool;   // Send all procedure
      sx_FIFOError { ExternalAccessible := 'False'; ExternalVisible := 'False'; ExternalWritable := 'False'} : Bool;   // FIFO error
      sx_FIFOWarning { ExternalAccessible := 'False'; ExternalVisible := 'False'; ExternalWritable := 'False'} : Bool;   // FIFO warning
      sx_ItemErrorBlockError { ExternalAccessible := 'False'; ExternalVisible := 'False'; ExternalWritable := 'False'} : Bool;   // Item error block error
      sx_ItemErrorBlockWarning { ExternalAccessible := 'False'; ExternalVisible := 'False'; ExternalWritable := 'False'} : Bool;   // Item error block warning
      sx_ItemStatusBlockError { ExternalAccessible := 'False'; ExternalVisible := 'False'; ExternalWritable := 'False'} : Bool;   // Item status block error
      sx_ItemStatusBlockWarning { ExternalAccessible := 'False'; ExternalVisible := 'False'; ExternalWritable := 'False'} : Bool;   // Item status block warning
   END_VAR


BEGIN
	(*
	----------------------------------------------------------------------------------------
	|                                                                                      |
	|  Copyright  2023             FORTNA Europe BV                                        |
	|  All Rights Reserved         Netherlands                                             |
	|                                                                                      |
	----------------------------------------------------------------------------------------
	Version history:
	Date        | Version   | Author       | Remark
	----------------------------------------------------------------------------------------
	30/03/2023  | 1.0       | M. Diebel   | Release TIA 17 | DHL Munich 2023
	13/03/2023  | 1.1       | S. Nieswiec  | Updated for new Baseline
	*)


	REGION 1 - Initialize message required signals

	    #sx_ItemErrorMessageReq := FALSE;
	    #sx_ItemStatusMessageReq := FALSE;

	    // On connection reestablish send last remembered status and error state ( status only when it's diffrent then 0 )
	    #s_R_TRIG_Connection(CLK := #ix_MFCConnected);

	    IF #s_R_TRIG_Connection.Q AND #si_ItemStatus <> 0
	    THEN
	        #sx_ItemStatusMessageReq := TRUE;
	    END_IF;

	    IF #s_R_TRIG_Connection.Q
	    THEN
	        #sx_ItemErrorMessageReq := TRUE;
	    END_IF;

	    // Prepare trigger on the collective reset signal.
	    #s_F_TRIG_SendAllErrors(CLK := #ix_SendAllErrorsState);

	    // When collective reset will go down, start send every equipment errors.
	    IF #s_F_TRIG_SendAllErrors.Q AND NOT #sx_SendAllProcedure
	    THEN
	        #ii_ErrorNumber := 0;
	        #sx_SendAllProcedure := TRUE;
	    END_IF;

	END_REGION

	REGION 2 - FIFO header status update

	    // Mode 'S' - FIFO register status update.
	    "FC_Fifo"(ic_Mode := 'S',
	              qUDT_Status => #ss_FIFOStatus,
	              qx_Error => #sx_FIFOError,
	              qx_Warning => #sx_FIFOWarning,
	              iqv_Data := #s_UDT_Message,
	              iqUDT_FifoHeader := #iq_UDT_FifoHeader,
	              iqv_DataBuffer := #iqs_FifoData);

	END_REGION

	REGION 3 - Prepare message data

	    // When there is no reset errors command, update status and errors.
	    IF NOT #ix_CollectiveReset
	        AND NOT #ss_FIFOStatus.FifoPreFull
	    THEN
	        // Status
	        IF (#i_UDT_CPGStatus.Status <> #s_UDT_CPGOld.Status OR (#sx_SendAllProcedure AND #ii_ErrorNumber = 0))
	        THEN
	            #sx_ItemStatusMessageReq := TRUE;
	            #si_ItemStatus := #i_UDT_CPGStatus.Status;
	            #s_UDT_CPGOld.Status := #i_UDT_CPGStatus.Status;
	        END_IF;


	        // Check which specific status changed, prepare code, change state and write new status into the old one.
	        IF (#i_UDT_CPGStatus.Specific.PowerSuppliesError <> #s_UDT_CPGOld.Specific.PowerSuppliesError AND NOT #sx_SendAllProcedure)
	            OR (#sx_SendAllProcedure AND #ii_ErrorNumber = 0)
	        THEN
	            #sdi_Code := "DB_MFC_ErrorCode".CPG.PowerSuppliesError;
	            #si_State := BOOL_TO_INT(#i_UDT_CPGStatus.Specific.PowerSuppliesError);
	            #s_UDT_CPGOld.Specific.PowerSuppliesError := #i_UDT_CPGStatus.Specific.PowerSuppliesError;
	            #sx_ItemErrorMessageReq := TRUE;
	            #sx_SendAllProcedure := FALSE;
	        END_IF;
	    END_IF;
	END_REGION

	REGION 4 - Write message components to the item error structure

	    #s_UDT_ItemError.ItemNumber := #i_UDT_EquipmentNumber;
	    #s_UDT_ItemError.Error := #sdi_Code;
	    #s_UDT_ItemError.State := #si_State;
	    #s_UDT_ItemError.Masked := 1;

	END_REGION

	REGION 5 - Write message components to the item status structure

	    #s_UDT_ItemStatus.Group := #i_UDT_EquipmentNumber.Group;
	    #s_UDT_ItemStatus.Node := #i_UDT_EquipmentNumber.Node;
	    #s_UDT_ItemStatus.Status := #si_ItemStatus;

	END_REGION

	REGION 6 - Prepare messages to the MFC

	    // If item error message required signal is set, prepare the item error message.
	    IF (#sx_ItemErrorMessageReq)
	    THEN
	        #s_FB_ItemError(i_UDT_ItemErrorBody := #s_UDT_ItemError,
	                        ii_MessageGroup := 1,
	                        ix_FlagRetry := FALSE,
	                        idi_TimeSpan := 0,
	                        qx_Error => #sx_ItemErrorBlockError,
	                        qx_Warning => #sx_ItemErrorBlockWarning,
	                        iq_UDT_FifoHeader := #iq_UDT_FifoHeader,
	                        iqs_FifoData := #iqs_FifoData,
	                        iqdi_MessageSequenceNumber := #iqdi_MessageSequenceNumber);
	    END_IF;

	    // If item status message required signal is set, prepare the item error message.
	    IF (#sx_ItemStatusMessageReq)
	    THEN
	        #s_FB_ItemStatus(i_UDT_ItemStatusBody := #s_UDT_ItemStatus,
	                         ii_MessageGroup := 1,
	                         ix_FlagRetry := FALSE,
	                         idi_TimeSpan := 0,
	                         qx_Error => #sx_ItemStatusBlockError,
	                         qx_Warning => #sx_ItemStatusBlockWarning,
	                         iq_UDT_FifoHeader := #iq_UDT_FifoHeader,
	                         iqs_FifoData := #iqs_FifoData,
	                         iqdi_MessageSequenceNumber := #iqdi_MessageSequenceNumber);
	    END_IF;

	END_REGION

	REGION 7 - Write outputs

	    // Prepare collective output error.
	    #qx_Error :=
	    #sx_ItemErrorBlockError
	    OR #sx_ItemStatusBlockError
	    OR #sx_FIFOError;

	    // Prepare collective output warning.
	    #qx_Warning :=
	    #sx_ItemErrorBlockWarning
	    OR #sx_ItemStatusBlockWarning
	    OR #sx_FIFOWarning;

	END_REGION
END_FUNCTION_BLOCK

FUNCTION_BLOCK "FB_MFC_Visu_Error_User"
{ S7_Optimized_Access := 'TRUE' }
VERSION : 0.1
// ATTRIBUTES
// AUTO_NUMBER = True
// BLOCK_NUMBER = 147
// END_ATTRIBUTES
   VAR_INPUT
      ix_Error { ExternalAccessible := 'False'; ExternalVisible := 'False'; ExternalWritable := 'False'} : Bool;
      i_UDT_EquipmentNumber { ExternalAccessible := 'False'; ExternalVisible := 'False'; ExternalWritable := 'False'} : "UDT_EquipmentNumber";   // Item number
      ix_SendAllErrorsState { ExternalAccessible := 'False'; ExternalVisible := 'False'; ExternalWritable := 'False'} : Bool;   // True - update all the messages
      ix_MFCConnected { ExternalAccessible := 'False'; ExternalVisible := 'False'; ExternalWritable := 'False'} : Bool;   // True - A connection to the MFC has been established
      ix_CollectiveReset { ExternalAccessible := 'False'; ExternalVisible := 'False'; ExternalWritable := 'False'} : Bool;   // True - Collective reset command of all system controls
      idi_Code { ExternalAccessible := 'False'; ExternalVisible := 'False'; ExternalWritable := 'False'} : DInt;
   END_VAR

   VAR_OUTPUT
      qx_Error { ExternalAccessible := 'False'; ExternalVisible := 'False'; ExternalWritable := 'False'} : Bool;   // Block error
      qx_Warning { ExternalAccessible := 'False'; ExternalVisible := 'False'; ExternalWritable := 'False'} : Bool;   // Block warning
   END_VAR

   VAR_IN_OUT
      iq_UDT_FifoHeader : "UDT_FifoHeader";   // FIFO header
      iqs_FifoData : Array[*] of "UDT_MessageV2";   // FIFO data buffer
      iqdi_MessageSequenceNumber { ExternalAccessible := 'False'; ExternalVisible := 'False'; ExternalWritable := 'False'} : DInt;   // Message number
   END_VAR

   VAR
      s_FB_ItemError { ExternalAccessible := 'False'; ExternalVisible := 'False'; ExternalWritable := 'False'; S7_SetPoint := 'False'} : "FB_ItemError";   // Item error block's instance
      ss_FIFOStatus { ExternalAccessible := 'False'; ExternalVisible := 'False'; ExternalWritable := 'False'; S7_SetPoint := 'False'} : "UDT_FifoStatus";   // Status structure
      s_UDT_Message { ExternalAccessible := 'False'; ExternalVisible := 'False'; ExternalWritable := 'False'; S7_SetPoint := 'False'} : "UDT_MessageV2";   // Message
      s_UDT_ItemError { ExternalAccessible := 'False'; ExternalVisible := 'False'; ExternalWritable := 'False'; S7_SetPoint := 'False'} : "UDT_ItemError";   // Item error message body structure
      s_R_TRIG_Connection {InstructionName := 'R_TRIG'; LibVersion := '1.0'; ExternalAccessible := 'False'; ExternalVisible := 'False'; ExternalWritable := 'False'; S7_SetPoint := 'False'} : R_TRIG;   // Rising edge trigger connection reastablished
      s_F_TRIG_SendAllErrors {InstructionName := 'F_TRIG'; LibVersion := '1.0'; ExternalAccessible := 'False'; ExternalVisible := 'False'; ExternalWritable := 'False'; S7_SetPoint := 'False'} : F_TRIG;   // Falling edge trigger from signal send all errors
      sdi_Code { ExternalAccessible := 'False'; ExternalVisible := 'False'; ExternalWritable := 'False'} : DInt;   // Error code
      si_State { ExternalAccessible := 'False'; ExternalVisible := 'False'; ExternalWritable := 'False'} : Int;   // Error state
      sx_ItemErrorMessageReq { ExternalAccessible := 'False'; ExternalVisible := 'False'; ExternalWritable := 'False'} : Bool;   // Item error message required
      sx_SendAllProcedure { ExternalAccessible := 'False'; ExternalVisible := 'False'; ExternalWritable := 'False'} : Bool;   // Send all procedure
      sx_FIFOError { ExternalAccessible := 'False'; ExternalVisible := 'False'; ExternalWritable := 'False'} : Bool;   // FIFO error
      sx_FIFOWarning { ExternalAccessible := 'False'; ExternalVisible := 'False'; ExternalWritable := 'False'} : Bool;   // FIFO warning
      sx_ItemErrorBlockError { ExternalAccessible := 'False'; ExternalVisible := 'False'; ExternalWritable := 'False'} : Bool;   // Item error block error
      sx_ItemErrorBlockWarning { ExternalAccessible := 'False'; ExternalVisible := 'False'; ExternalWritable := 'False'} : Bool;   // Item error block warning
      sx_OldError { ExternalAccessible := 'False'; ExternalVisible := 'False'; ExternalWritable := 'False'} : Bool;
   END_VAR


BEGIN
	(*
	----------------------------------------------------------------------------------------
	|                                                                                      |
	|  Copyright  2023             FORTNA Europe BV                                        |
	|  All Rights Reserved         Netherlands                                             |
	|                                                                                      |
	----------------------------------------------------------------------------------------
	Version history:
	Date        | Version   | Author       | Remark
	29/01/2024  | 1.0       | M. Diebel   | Release TIA 17 | DHL Munich 2023
	13/03/2023  | 1.1       | S. Nieswiec  | Updated for new Baseline
	*)

	REGION 1 - Initialize message required signals

	    #sx_ItemErrorMessageReq := FALSE;

	    // On connection reestablish send last remembered status and error state ( status only when it's diffrent then 0 )
	    #s_R_TRIG_Connection(CLK := #ix_MFCConnected);

	    IF #s_R_TRIG_Connection.Q
	    THEN
	        #sx_ItemErrorMessageReq := TRUE;
	    END_IF;

	    // Prepare trigger on the collective reset signal.
	    #s_F_TRIG_SendAllErrors(CLK := #ix_SendAllErrorsState);

	    // When collective reset will go down, start send every equipment errors.
	    IF #s_F_TRIG_SendAllErrors.Q AND NOT #sx_SendAllProcedure
	    THEN
	        #sx_SendAllProcedure := TRUE;
	    END_IF;

	END_REGION

	REGION 2 - FIFO header status update

	    // Mode 'S' - FIFO register status update.
	    "FC_Fifo"(ic_Mode := 'S',
	              qUDT_Status => #ss_FIFOStatus,
	              qx_Error => #sx_FIFOError,
	              qx_Warning => #sx_FIFOWarning,
	              iqv_Data := #s_UDT_Message,
	              iqUDT_FifoHeader := #iq_UDT_FifoHeader,
	              iqv_DataBuffer := #iqs_FifoData);

	END_REGION

	REGION 3 - Prepare message data

	    // When there is no reset errors command, update status and errors.
	    IF NOT #ix_CollectiveReset
	        AND NOT #ss_FIFOStatus.FifoPreFull
	    THEN

	        // Check which specific status changed, prepare code, change state and write new status into the old one.
	        IF (#ix_Error <> #sx_OldError AND NOT #sx_SendAllProcedure)
	            OR (#sx_SendAllProcedure)
	        THEN
	            #sdi_Code := #idi_Code;
	            #si_State := BOOL_TO_INT(#ix_Error);
	            #sx_OldError := #ix_Error;
	            #sx_ItemErrorMessageReq := TRUE;
	            #sx_SendAllProcedure := FALSE;
	        END_IF;

	    END_IF;
	END_REGION

	REGION 4 - Write message components to the item error structure

	    #s_UDT_ItemError.ItemNumber := #i_UDT_EquipmentNumber;
	    #s_UDT_ItemError.Error := #sdi_Code;
	    #s_UDT_ItemError.State := #si_State;
	    #s_UDT_ItemError.Masked := 1;

	END_REGION

	REGION 6 - Prepare messages to the MFC

	    // If item error message required signal is set, prepare the item error message.
	    IF (#sx_ItemErrorMessageReq)
	    THEN
	        #s_FB_ItemError(i_UDT_ItemErrorBody := #s_UDT_ItemError,
	                        ii_MessageGroup := 1,
	                        ix_FlagRetry := FALSE,
	                        idi_TimeSpan := 0,
	                        qx_Error => #sx_ItemErrorBlockError,
	                        qx_Warning => #sx_ItemErrorBlockWarning,
	                        iq_UDT_FifoHeader := #iq_UDT_FifoHeader,
	                        iqs_FifoData := #iqs_FifoData,
	                        iqdi_MessageSequenceNumber := #iqdi_MessageSequenceNumber);
	    END_IF;

	END_REGION

	REGION 7 - Write outputs

	    // Prepare collective output error.
	    #qx_Error :=
	    #sx_ItemErrorBlockError
	    OR #sx_FIFOError;

	    // Prepare collective output warning.
	    #qx_Warning :=
	    #sx_ItemErrorBlockWarning
	    OR #sx_FIFOWarning;

	END_REGION
END_FUNCTION_BLOCK

FUNCTION_BLOCK "FB_MFC_Visu_EncoderValue_Status"
{ S7_Optimized_Access := 'TRUE' }
VERSION : 0.1
// ATTRIBUTES
// AUTO_NUMBER = True
// BLOCK_NUMBER = 146
// END_ATTRIBUTES
   VAR_INPUT
      i_UDT_EncoderStatus { ExternalAccessible := 'False'; ExternalVisible := 'False'; ExternalWritable := 'False'} : "UDT_EncoderStatusV2";   // EncoderStatus status structure
      i_UDT_EquipmentNumber { ExternalAccessible := 'False'; ExternalVisible := 'False'; ExternalWritable := 'False'} : "UDT_EquipmentNumber";   // Item number
      ix_SendAllErrorsState { ExternalAccessible := 'False'; ExternalVisible := 'False'; ExternalWritable := 'False'} : Bool;   // True - update all the messages
      ix_MFCConnected { ExternalAccessible := 'False'; ExternalVisible := 'False'; ExternalWritable := 'False'} : Bool;   // True - A connection to the MFC has been established
      ix_CollectiveReset { ExternalAccessible := 'False'; ExternalVisible := 'False'; ExternalWritable := 'False'} : Bool;   // True - Collective reset command of all system controls
   END_VAR

   VAR_OUTPUT
      qx_Error { ExternalAccessible := 'False'; ExternalVisible := 'False'; ExternalWritable := 'False'} : Bool;   // Block error
      qx_Warning { ExternalAccessible := 'False'; ExternalVisible := 'False'; ExternalWritable := 'False'} : Bool;   // Block warning
   END_VAR

   VAR_IN_OUT
      iq_UDT_FifoHeader : "UDT_FifoHeader";   // FIFO header
      iqs_FifoData : Array[*] of "UDT_MessageV2";   // FIFO data buffer
      iqdi_MessageSequenceNumber { ExternalAccessible := 'False'; ExternalVisible := 'False'; ExternalWritable := 'False'} : DInt;   // Message number
   END_VAR

   VAR
      s_FB_ItemError { ExternalAccessible := 'False'; ExternalVisible := 'False'; ExternalWritable := 'False'; S7_SetPoint := 'False'} : "FB_ItemError";   // Item error block's instance
      s_FB_ItemStatus { ExternalAccessible := 'False'; ExternalVisible := 'False'; ExternalWritable := 'False'; S7_SetPoint := 'False'} : "FB_ItemStatus";   // Item status block's instance
      ss_FIFOStatus { ExternalAccessible := 'False'; ExternalVisible := 'False'; ExternalWritable := 'False'; S7_SetPoint := 'False'} : "UDT_FifoStatus";   // Status structure
      s_UDT_Message { ExternalAccessible := 'False'; ExternalVisible := 'False'; ExternalWritable := 'False'; S7_SetPoint := 'False'} : "UDT_MessageV2";   // Message
      s_UDT_EncoderOld { ExternalAccessible := 'False'; ExternalVisible := 'False'; ExternalWritable := 'False'; S7_SetPoint := 'False'} : "UDT_EncoderStatusV2";   // Encoder  status structure
      s_UDT_ItemError { ExternalAccessible := 'False'; ExternalVisible := 'False'; ExternalWritable := 'False'; S7_SetPoint := 'False'} : "UDT_ItemError";   // Item error message body structure
      s_UDT_ItemStatus { ExternalAccessible := 'False'; ExternalVisible := 'False'; ExternalWritable := 'False'; S7_SetPoint := 'False'} : "UDT_ItemStatus";   // Item status message body structure
      s_R_TRIG_Connection {InstructionName := 'R_TRIG'; LibVersion := '1.0'; ExternalAccessible := 'False'; ExternalVisible := 'False'; ExternalWritable := 'False'; S7_SetPoint := 'False'} : R_TRIG;   // Rising edge trigger connection reastablished
      s_F_TRIG_SendAllErrors {InstructionName := 'F_TRIG'; LibVersion := '1.0'; ExternalAccessible := 'False'; ExternalVisible := 'False'; ExternalWritable := 'False'; S7_SetPoint := 'False'} : F_TRIG;   // Falling edge trigger from signal send all errors
      sdi_Code { ExternalAccessible := 'False'; ExternalVisible := 'False'; ExternalWritable := 'False'} : DInt;   // Error code
      si_ItemStatus { ExternalAccessible := 'False'; ExternalVisible := 'False'; ExternalWritable := 'False'} : Int;   // Item status
      ii_ErrorNumber { ExternalAccessible := 'False'; ExternalVisible := 'False'; ExternalWritable := 'False'} : Int;   // Counter Error Number
      si_State { ExternalAccessible := 'False'; ExternalVisible := 'False'; ExternalWritable := 'False'} : Int;   // Error state
      sx_ItemErrorMessageReq { ExternalAccessible := 'False'; ExternalVisible := 'False'; ExternalWritable := 'False'} : Bool;   // Item error message required
      sx_ItemStatusMessageReq { ExternalAccessible := 'False'; ExternalVisible := 'False'; ExternalWritable := 'False'} : Bool;   // Item status message required
      sx_SendAllProcedure { ExternalAccessible := 'False'; ExternalVisible := 'False'; ExternalWritable := 'False'} : Bool;   // Send all procedure
      sx_FIFOError { ExternalAccessible := 'False'; ExternalVisible := 'False'; ExternalWritable := 'False'} : Bool;   // FIFO error
      sx_FIFOWarning { ExternalAccessible := 'False'; ExternalVisible := 'False'; ExternalWritable := 'False'} : Bool;   // FIFO warning
      sx_ItemErrorBlockError { ExternalAccessible := 'False'; ExternalVisible := 'False'; ExternalWritable := 'False'} : Bool;   // Item error block error
      sx_ItemErrorBlockWarning { ExternalAccessible := 'False'; ExternalVisible := 'False'; ExternalWritable := 'False'} : Bool;   // Item error block warning
      sx_ItemStatusBlockError { ExternalAccessible := 'False'; ExternalVisible := 'False'; ExternalWritable := 'False'} : Bool;   // Item status block error
      sx_ItemStatusBlockWarning { ExternalAccessible := 'False'; ExternalVisible := 'False'; ExternalWritable := 'False'} : Bool;   // Item status block warning
   END_VAR


BEGIN
	(*
	----------------------------------------------------------------------------------------
	|                                                                                      |
	|  Copyright  2023             FORTNA Europe BV                                        |
	|  All Rights Reserved         Netherlands                                             |
	|                                                                                      |
	----------------------------------------------------------------------------------------
	Version history:
	Date        | Version   | Author       | Remark
	----------------------------------------------------------------------------------------
	29/03/2023  | 1.0       | M. Diebel   | Release TIA 17 | DHL Munich 2023
	13/03/2023  | 1.1       | S. Nieswiec  | Updated for new Baseline
	*)


	REGION 1 - Initialize message required signals

	    #sx_ItemErrorMessageReq := FALSE;

	    // On connection reestablish send last remembered status and error state ( status only when it's diffrent then 0 )
	    #s_R_TRIG_Connection(CLK := #ix_MFCConnected);


	    IF #s_R_TRIG_Connection.Q
	    THEN
	        #sx_ItemErrorMessageReq := TRUE;
	    END_IF;

	    // Prepare trigger on the collective reset signal.
	    #s_F_TRIG_SendAllErrors(CLK := #ix_SendAllErrorsState);

	    // When collective reset will go down, start send every equipment errors.
	    IF #s_F_TRIG_SendAllErrors.Q AND NOT #sx_SendAllProcedure
	    THEN
	        #ii_ErrorNumber := 0;
	        #sx_SendAllProcedure := TRUE;
	    END_IF;

	END_REGION

	REGION 2 - FIFO header status update

	    // Mode 'S' - FIFO register status update.
	    "FC_Fifo"(ic_Mode := 'S',
	              qUDT_Status => #ss_FIFOStatus,
	              qx_Error => #sx_FIFOError,
	              qx_Warning => #sx_FIFOWarning,
	              iqv_Data := #s_UDT_Message,
	              iqUDT_FifoHeader := #iq_UDT_FifoHeader,
	              iqv_DataBuffer := #iqs_FifoData);

	END_REGION

	REGION 3 - Prepare message data

	    IF NOT #ix_CollectiveReset
	        AND NOT #ss_FIFOStatus.FifoPreFull
	    THEN

	        // Check which specific status changed, prepare code, change state and write new status into the old one.
	        IF (#i_UDT_EncoderStatus.InvalidValue <> #s_UDT_EncoderOld.InvalidValue AND NOT #sx_SendAllProcedure)
	            OR (#sx_SendAllProcedure AND #ii_ErrorNumber = 0)
	        THEN
	            #sdi_Code := "DB_MFC_ErrorCode".Encoder.InvalidValue;
	            #si_State := BOOL_TO_INT(#i_UDT_EncoderStatus.InvalidValue);
	            #s_UDT_EncoderOld.InvalidValue := #i_UDT_EncoderStatus.InvalidValue;
	            #sx_ItemErrorMessageReq := TRUE;
	            #ii_ErrorNumber += 1;
	        ELSIF (#i_UDT_EncoderStatus.RunningFeedbackError <> #s_UDT_EncoderOld.RunningFeedbackError AND NOT #sx_SendAllProcedure)
	            OR (#sx_SendAllProcedure AND #ii_ErrorNumber = 1)
	        THEN
	            #sdi_Code := "DB_MFC_ErrorCode".Encoder.RunningFeedbackError;
	            #si_State := BOOL_TO_INT(#i_UDT_EncoderStatus.RunningFeedbackError);
	            #s_UDT_EncoderOld.RunningFeedbackError := #i_UDT_EncoderStatus.RunningFeedbackError;
	            #sx_ItemErrorMessageReq := TRUE;
	            #sx_SendAllProcedure := FALSE;
	            #ii_ErrorNumber += 1;
	        END_IF;
	    END_IF;

	END_REGION

	REGION 4 - Write message components to the item error structure

	    #s_UDT_ItemError.ItemNumber := #i_UDT_EquipmentNumber;
	    #s_UDT_ItemError.Error := #sdi_Code;
	    #s_UDT_ItemError.State := #si_State;
	    #s_UDT_ItemError.Masked := 1;

	END_REGION


	REGION 6 - Prepare messages to the MFC

	    // If item error message required signal is set, prepare the item error message.
	    IF (#sx_ItemErrorMessageReq)
	    THEN
	        #s_FB_ItemError(i_UDT_ItemErrorBody := #s_UDT_ItemError,
	                        ii_MessageGroup := 1,
	                        ix_FlagRetry := FALSE,
	                        idi_TimeSpan := 0,
	                        qx_Error => #sx_ItemErrorBlockError,
	                        qx_Warning => #sx_ItemErrorBlockWarning,
	                        iq_UDT_FifoHeader := #iq_UDT_FifoHeader,
	                        iqs_FifoData := #iqs_FifoData,
	                        iqdi_MessageSequenceNumber := #iqdi_MessageSequenceNumber);
	    END_IF;


	END_REGION

	REGION 7 - Write outputs

	    // Prepare collective output error.
	    #qx_Error :=
	    #sx_ItemErrorBlockError
	    OR #sx_FIFOError;

	    // Prepare collective output warning.
	    #qx_Warning :=
	    #sx_ItemErrorBlockWarning
	    OR #sx_FIFOWarning;

	END_REGION



END_FUNCTION_BLOCK

FUNCTION_BLOCK "FB_MFC_Visu_DMC_Status"
{ S7_Optimized_Access := 'TRUE' }
VERSION : 0.1
// ATTRIBUTES
// AUTO_NUMBER = True
// BLOCK_NUMBER = 145
// END_ATTRIBUTES
   VAR_INPUT
      ix_SendAllErrorsState { ExternalAccessible := 'False'; ExternalVisible := 'False'; ExternalWritable := 'False'} : Bool;   // True - update all the messages
      ix_MFCConnected { ExternalAccessible := 'False'; ExternalVisible := 'False'; ExternalWritable := 'False'} : Bool;   // True - A connection to the MFC has been established
      ix_CollectiveReset { ExternalAccessible := 'False'; ExternalVisible := 'False'; ExternalWritable := 'False'} : Bool;   // True - Collective reset command of all system controls
      i_UDT_DMCStatus { ExternalAccessible := 'False'; ExternalVisible := 'False'; ExternalWritable := 'False'} : "UDT_DimensionsCheckStatusV2";   // Dimensions check status error structure
      i_UDT_EquipmentNumber { ExternalAccessible := 'False'; ExternalVisible := 'False'; ExternalWritable := 'False'} : "UDT_EquipmentNumber";   // Item number
   END_VAR

   VAR_OUTPUT
      qx_Error { ExternalAccessible := 'False'; ExternalVisible := 'False'; ExternalWritable := 'False'} : Bool;   // Block error
      qx_Warning { ExternalAccessible := 'False'; ExternalVisible := 'False'; ExternalWritable := 'False'} : Bool;   // Block warning
   END_VAR

   VAR_IN_OUT
      iq_UDT_FifoHeader : "UDT_FifoHeader";   // FIFO header
      iqs_FifoData : Array[*] of "UDT_MessageV2";   // FIFO data buffer
      iqdi_MessageSequenceNumber { ExternalAccessible := 'False'; ExternalVisible := 'False'; ExternalWritable := 'False'} : DInt;   // Message number
   END_VAR

   VAR
      s_FB_ItemError { ExternalAccessible := 'False'; ExternalVisible := 'False'; ExternalWritable := 'False'; S7_SetPoint := 'False'} : "FB_ItemError";   // Item error block's instance
      s_FB_ItemStatus { ExternalAccessible := 'False'; ExternalVisible := 'False'; ExternalWritable := 'False'; S7_SetPoint := 'False'} : "FB_ItemStatus";   // Item status block's instance
      s_UDT_ItemError { ExternalAccessible := 'False'; ExternalVisible := 'False'; ExternalWritable := 'False'; S7_SetPoint := 'False'} : "UDT_ItemError";   // Item error message body structure
      s_UDT_ItemStatus { ExternalAccessible := 'False'; ExternalVisible := 'False'; ExternalWritable := 'False'; S7_SetPoint := 'False'} : "UDT_ItemStatus";   // Item status message body structure
      s_UDT_Message { ExternalAccessible := 'False'; ExternalVisible := 'False'; ExternalWritable := 'False'; S7_SetPoint := 'False'} : "UDT_BytesMessage";   // Message
      s_UDT_DMCOld { ExternalAccessible := 'False'; ExternalVisible := 'False'; ExternalWritable := 'False'; S7_SetPoint := 'False'} : "UDT_DimensionsCheckStatusV2";   // DMC old status structure
      s_UDT_FIFOStatus { ExternalAccessible := 'False'; ExternalVisible := 'False'; ExternalWritable := 'False'; S7_SetPoint := 'False'} : "UDT_FifoStatus";   // FIFO status structure
      ss_FIFOStatus { ExternalAccessible := 'False'; ExternalVisible := 'False'; ExternalWritable := 'False'; S7_SetPoint := 'False'} : "UDT_FifoStatus";   // Status structure
      s_R_TRIG_Connection {InstructionName := 'R_TRIG'; LibVersion := '1.0'; ExternalAccessible := 'False'; ExternalVisible := 'False'; ExternalWritable := 'False'; S7_SetPoint := 'False'} : R_TRIG;   // Rising edge trigger connection reastablished
      s_F_TRIG_SendAllErrors {InstructionName := 'F_TRIG'; LibVersion := '1.0'; ExternalAccessible := 'False'; ExternalVisible := 'False'; ExternalWritable := 'False'; S7_SetPoint := 'False'} : F_TRIG;   // Falling edge trigger from signal send all errors
      slr_RunningTimeMS { ExternalAccessible := 'False'; ExternalVisible := 'False'; ExternalWritable := 'False'} : LReal;   // Conveyor running time [ms]
      sdi_DistanceTraveled { ExternalAccessible := 'False'; ExternalVisible := 'False'; ExternalWritable := 'False'} : DInt;   // Distance traveled by conveyor
      sdi_StartStop { ExternalAccessible := 'False'; ExternalVisible := 'False'; ExternalWritable := 'False'} : DInt;   // Value of change conveyor state from start to stop and from stop to start
      sdi_Code { ExternalAccessible := 'False'; ExternalVisible := 'False'; ExternalWritable := 'False'} : DInt;   // Error code
      sdi_RunningTime { ExternalAccessible := 'False'; ExternalVisible := 'False'; ExternalWritable := 'False'} : DInt;   // Conveyor running time [s]
      si_ItemStatus { ExternalAccessible := 'False'; ExternalVisible := 'False'; ExternalWritable := 'False'} : Int;   // Item status
      si_State { ExternalAccessible := 'False'; ExternalVisible := 'False'; ExternalWritable := 'False'} : Int;   // Error state
      ii_ErrorNumber { ExternalAccessible := 'False'; ExternalVisible := 'False'; ExternalWritable := 'False'} : Int;   // Counter Error Number
      sx_ItemErrorMessageReq { ExternalAccessible := 'False'; ExternalVisible := 'False'; ExternalWritable := 'False'} : Bool;   // Item error message required
      sx_ItemStatusMessageReq { ExternalAccessible := 'False'; ExternalVisible := 'False'; ExternalWritable := 'False'} : Bool;   // Item status message required
      sx_ItemErrorBlockError { ExternalAccessible := 'False'; ExternalVisible := 'False'; ExternalWritable := 'False'} : Bool;   // Item error block error
      sx_ItemStatusBlockError { ExternalAccessible := 'False'; ExternalVisible := 'False'; ExternalWritable := 'False'} : Bool;   // Item status block error
      sx_FIFOError { ExternalAccessible := 'False'; ExternalVisible := 'False'; ExternalWritable := 'False'} : Bool;   // FIFO error
      sx_FIFOWarning { ExternalAccessible := 'False'; ExternalVisible := 'False'; ExternalWritable := 'False'} : Bool;   // FIFO warning
      sx_MaintenanceCounterBlockError { ExternalAccessible := 'False'; ExternalVisible := 'False'; ExternalWritable := 'False'} : Bool;   // Maintenance counter block error
      sx_ItemStatusBlockWarning { ExternalAccessible := 'False'; ExternalVisible := 'False'; ExternalWritable := 'False'} : Bool;   // Item status block warning
      sx_ItemErrorBlockWarning { ExternalAccessible := 'False'; ExternalVisible := 'False'; ExternalWritable := 'False'} : Bool;   // Item error block warning
      sx_MaintenanceCounterBlockWarning { ExternalAccessible := 'False'; ExternalVisible := 'False'; ExternalWritable := 'False'} : Bool;   // Maintenance counter block warning
      sx_SendAllProcedure { ExternalAccessible := 'False'; ExternalVisible := 'False'; ExternalWritable := 'False'} : Bool;   // Send all procedure
   END_VAR


BEGIN
	(*
	----------------------------------------------------------------------------------------
	|                                                                                      |
	|  Copyright  2023             FORTNA Europe BV                                        |
	|  All Rights Reserved         Netherlands                                             |
	|                                                                                      |
	----------------------------------------------------------------------------------------
	Version history:
	Date        | Version   | Author       | Remark
	----------------------------------------------------------------------------------------
	03/01/2023  | 1.0       | S. Nikodem   | Release TIA 17 | DHL Munich 2023
	13/03/2023  | 1.1       | S. Nieswiec  | Updated for new Baseline
	*)

	REGION 1 - Initialize message required signals

	    #sx_ItemErrorMessageReq := FALSE;
	    #sx_ItemStatusMessageReq := FALSE;

	    // On connection reestablish send last remembered status and error state ( status only when it's diffrent then 0 )
	    #s_R_TRIG_Connection(CLK := #ix_MFCConnected);

	    IF #s_R_TRIG_Connection.Q AND #si_ItemStatus <> 0
	    THEN
	        #sx_ItemStatusMessageReq := TRUE;
	    END_IF;

	    IF #s_R_TRIG_Connection.Q
	    THEN
	        #sx_ItemErrorMessageReq := TRUE;
	    END_IF;

	    // Prepare trigger on the collective reset signal.
	    #s_F_TRIG_SendAllErrors(CLK := #ix_SendAllErrorsState);

	    // When collective reset will go down, start send every equipment errors.
	    IF #s_F_TRIG_SendAllErrors.Q AND NOT #sx_SendAllProcedure
	    THEN
	        #ii_ErrorNumber := 0;
	        #sx_SendAllProcedure := TRUE;
	    END_IF;

	END_REGION

	REGION 2 - FIFO header status update

	    // Mode 'S' - FIFO register status update.
	    "FC_Fifo"(ic_Mode := 'S',
	              qUDT_Status => #ss_FIFOStatus,
	              qx_Error => #sx_FIFOError,
	              qx_Warning => #sx_FIFOWarning,
	              iqv_Data := #s_UDT_Message,
	              iqUDT_FifoHeader := #iq_UDT_FifoHeader,
	              iqv_DataBuffer := #iqs_FifoData);

	END_REGION

	REGION 3 - Prepare message data

	    // When there is no reset errors command, update status and errors.
	    IF NOT #ix_CollectiveReset
	        AND NOT #ss_FIFOStatus.FifoPreFull
	    THEN

	        IF (#i_UDT_DMCStatus.Status <> #s_UDT_DMCOld.Status OR (#sx_SendAllProcedure AND #ii_ErrorNumber = 0))
	        THEN
	            #sx_ItemStatusMessageReq := TRUE;
	            #si_ItemStatus := #i_UDT_DMCStatus.Status;
	            #s_UDT_DMCOld.Status := #i_UDT_DMCStatus.Status;
	        END_IF;

	        // Check which specific status changed, prepare code, change state and write new status into the old one.
	        IF (#i_UDT_DMCStatus.Specific.ParcelTooLongError <> #s_UDT_DMCOld.Specific.ParcelTooLongError AND NOT #sx_SendAllProcedure)
	            OR (#sx_SendAllProcedure AND #ii_ErrorNumber = 0)
	        THEN
	            #sdi_Code := "DB_MFC_ErrorCode".DMC.ParcelTooLong;
	            #si_State := BOOL_TO_INT(#i_UDT_DMCStatus.Specific.ParcelTooLongError);
	            #s_UDT_DMCOld.Specific.ParcelTooLongError := #i_UDT_DMCStatus.Specific.ParcelTooLongError;
	            #sx_ItemErrorMessageReq := TRUE;
	            #ii_ErrorNumber += 1;
	        ELSIF (#i_UDT_DMCStatus.Specific.ParcelTooShortError <> #s_UDT_DMCOld.Specific.ParcelTooShortError AND NOT #sx_SendAllProcedure)
	            OR (#sx_SendAllProcedure AND #ii_ErrorNumber = 1)
	        THEN
	            #sdi_Code := "DB_MFC_ErrorCode".DMC.ParcelTooShort;
	            #si_State := BOOL_TO_INT(#i_UDT_DMCStatus.Specific.ParcelTooShortError);
	            #s_UDT_DMCOld.Specific.ParcelTooShortError := #i_UDT_DMCStatus.Specific.ParcelTooShortError;
	            #sx_ItemErrorMessageReq := TRUE;
	            #ii_ErrorNumber += 1;
	        ELSIF (#i_UDT_DMCStatus.Specific.ParcelTooHighError <> #s_UDT_DMCOld.Specific.ParcelTooHighError AND NOT #sx_SendAllProcedure)
	            OR (#sx_SendAllProcedure AND #ii_ErrorNumber = 2)
	        THEN
	            #sdi_Code := "DB_MFC_ErrorCode".DMC.ParcelTooHigh;
	            #si_State := BOOL_TO_INT(#i_UDT_DMCStatus.Specific.ParcelTooHighError);
	            #s_UDT_DMCOld.Specific.ParcelTooHighError := #i_UDT_DMCStatus.Specific.ParcelTooHighError;
	            #sx_ItemErrorMessageReq := TRUE;
	            #ii_ErrorNumber += 1;
	        ELSIF (#i_UDT_DMCStatus.Specific.ParcelTooLowError <> #s_UDT_DMCOld.Specific.ParcelTooLowError AND NOT #sx_SendAllProcedure)
	            OR (#sx_SendAllProcedure AND #ii_ErrorNumber = 3)
	        THEN
	            #sdi_Code := "DB_MFC_ErrorCode".DMC.ParcelTooLow;
	            #si_State := BOOL_TO_INT(#i_UDT_DMCStatus.Specific.ParcelTooLowError);
	            #s_UDT_DMCOld.Specific.ParcelTooLowError := #i_UDT_DMCStatus.Specific.ParcelTooLowError;
	            #sx_ItemErrorMessageReq := TRUE;
	            #ii_ErrorNumber += 1;
	        ELSIF (#i_UDT_DMCStatus.Specific.ParcelTooWideError <> #s_UDT_DMCOld.Specific.ParcelTooWideError AND NOT #sx_SendAllProcedure)
	            OR (#sx_SendAllProcedure AND #ii_ErrorNumber = 4)
	        THEN
	            #sdi_Code := "DB_MFC_ErrorCode".DMC.ParcelTooWide;
	            #si_State := BOOL_TO_INT(#i_UDT_DMCStatus.Specific.ParcelTooWideError);
	            #s_UDT_DMCOld.Specific.ParcelTooWideError := #i_UDT_DMCStatus.Specific.ParcelTooWideError;
	            #sx_ItemErrorMessageReq := TRUE;
	            #ii_ErrorNumber += 1;
	        ELSIF (#i_UDT_DMCStatus.Specific.ParcelTooNarrowError <> #s_UDT_DMCOld.Specific.ParcelTooNarrowError AND NOT #sx_SendAllProcedure)
	            OR (#sx_SendAllProcedure AND #ii_ErrorNumber = 5)
	        THEN
	            #sdi_Code := "DB_MFC_ErrorCode".DMC.ParcelTooNarrow;
	            #si_State := BOOL_TO_INT(#i_UDT_DMCStatus.Specific.ParcelTooNarrowError);
	            #s_UDT_DMCOld.Specific.ParcelTooNarrowError := #i_UDT_DMCStatus.Specific.ParcelTooNarrowError;
	            #sx_ItemErrorMessageReq := TRUE;
	            #ii_ErrorNumber += 1;
	        ELSIF (#i_UDT_DMCStatus.Specific.IncorrectParcelOrientationError <> #s_UDT_DMCOld.Specific.IncorrectParcelOrientationError AND NOT #sx_SendAllProcedure)
	            OR (#sx_SendAllProcedure AND #ii_ErrorNumber = 6)
	        THEN
	            #sdi_Code := "DB_MFC_ErrorCode".DMC.IncorrectParcelOrientationError;
	            #si_State := BOOL_TO_INT(#i_UDT_DMCStatus.Specific.IncorrectParcelOrientationError);
	            #s_UDT_DMCOld.Specific.IncorrectParcelOrientationError := #i_UDT_DMCStatus.Specific.IncorrectParcelOrientationError;
	            #sx_ItemErrorMessageReq := TRUE;
	            #ii_ErrorNumber += 1;
	        ELSIF (#i_UDT_DMCStatus.Specific.GeneralError <> #s_UDT_DMCOld.Specific.GeneralError AND NOT #sx_SendAllProcedure)
	            OR (#sx_SendAllProcedure AND #ii_ErrorNumber = 7)
	        THEN
	            #sdi_Code := "DB_MFC_ErrorCode".DMC.GeneralError;
	            #si_State := BOOL_TO_INT(#i_UDT_DMCStatus.Specific.GeneralError);
	            #s_UDT_DMCOld.Specific.GeneralError := #i_UDT_DMCStatus.Specific.GeneralError;
	            #sx_ItemErrorMessageReq := TRUE;
	            #ii_ErrorNumber += 1;
	        END_IF;

	    END_IF;

	END_REGION

	REGION 4 - Write message components to the item error structure

	    #s_UDT_ItemError.ItemNumber := #i_UDT_EquipmentNumber;
	    #s_UDT_ItemError.Error := #sdi_Code;
	    #s_UDT_ItemError.State := #si_State;
	    #s_UDT_ItemError.Masked := 1;

	END_REGION

	REGION 5 - Write message components to the item status structure

	    // Adjust library statuses into the client one.
	    // To check later
	    // Status:
	    //     19 – Running
	    //     21 - EnergySave
	    //     0 - Stopped
	    //     23 - DimensionError
	    //     3 – SafetyStop


	    #s_UDT_ItemStatus.Group := #i_UDT_EquipmentNumber.Group;
	    #s_UDT_ItemStatus.Node := #i_UDT_EquipmentNumber.Node;
	    #s_UDT_ItemStatus.Status := #si_ItemStatus;

	END_REGION

	REGION 6 - Prepare messages to the MFC

	    // If item error message required signal is set, prepare the item error message.
	    IF (#sx_ItemErrorMessageReq)
	    THEN
	        #s_FB_ItemError(i_UDT_ItemErrorBody := #s_UDT_ItemError,
	                        ii_MessageGroup := 1,
	                        ix_FlagRetry := FALSE,
	                        idi_TimeSpan := 0,
	                        qx_Error => #sx_ItemErrorBlockError,
	                        qx_Warning => #sx_ItemErrorBlockWarning,
	                        iq_UDT_FifoHeader := #iq_UDT_FifoHeader,
	                        iqs_FifoData := #iqs_FifoData,
	                        iqdi_MessageSequenceNumber := #iqdi_MessageSequenceNumber);
	    END_IF;

	    // If item status message required signal is set, prepare the item error message.
	    IF (#sx_ItemStatusMessageReq)
	    THEN
	        #s_FB_ItemStatus(i_UDT_ItemStatusBody := #s_UDT_ItemStatus,
	                         ii_MessageGroup := 1,
	                         ix_FlagRetry := FALSE,
	                         idi_TimeSpan := 0,
	                         qx_Error => #sx_ItemStatusBlockError,
	                         qx_Warning => #sx_ItemStatusBlockWarning,
	                         iq_UDT_FifoHeader := #iq_UDT_FifoHeader,
	                         iqs_FifoData := #iqs_FifoData,
	                         iqdi_MessageSequenceNumber := #iqdi_MessageSequenceNumber);
	    END_IF;

	END_REGION

	REGION 7 - Write outputs

	    // Prepare collective output error.
	    #qx_Error :=
	    #sx_ItemErrorBlockError
	    OR #sx_ItemStatusBlockError
	    OR #sx_MaintenanceCounterBlockError
	    OR #sx_FIFOError;

	    // Prepare collective output warning.
	    #qx_Warning :=
	    #sx_ItemErrorBlockWarning
	    OR #sx_ItemStatusBlockWarning
	    OR #sx_MaintenanceCounterBlockWarning
	    OR #sx_FIFOWarning;

	END_REGION
END_FUNCTION_BLOCK

FUNCTION_BLOCK "FB_MFC_Visu_DimensionsCheck_Status"
{ S7_Optimized_Access := 'TRUE' }
VERSION : 0.1
// ATTRIBUTES
// AUTO_NUMBER = True
// BLOCK_NUMBER = 144
// END_ATTRIBUTES
   VAR_INPUT
      i_UDT_DimensionsCheckStatus { ExternalAccessible := 'False'; ExternalVisible := 'False'; ExternalWritable := 'False'} : "UDT_DimensionsCheckStatusV2";   // DimensionChceck status structure
      i_UDT_EquipmentNumber { ExternalAccessible := 'False'; ExternalVisible := 'False'; ExternalWritable := 'False'} : "UDT_EquipmentNumber";   // Item number
      ix_SendAllErrorsState { ExternalAccessible := 'False'; ExternalVisible := 'False'; ExternalWritable := 'False'} : Bool;   // True - update all the messages
      ix_MFCConnected { ExternalAccessible := 'False'; ExternalVisible := 'False'; ExternalWritable := 'False'} : Bool;   // True - A connection to the MFC has been established
      ix_CollectiveReset { ExternalAccessible := 'False'; ExternalVisible := 'False'; ExternalWritable := 'False'} : Bool;   // True - Collective reset command of all system controls
   END_VAR

   VAR_OUTPUT
      qx_Error { ExternalAccessible := 'False'; ExternalVisible := 'False'; ExternalWritable := 'False'} : Bool;   // Block error
      qx_Warning { ExternalAccessible := 'False'; ExternalVisible := 'False'; ExternalWritable := 'False'} : Bool;   // Block warning
   END_VAR

   VAR_IN_OUT
      iq_UDT_FifoHeader : "UDT_FifoHeader";   // FIFO header
      iqs_FifoData : Array[*] of "UDT_MessageV2";   // FIFO data buffer
      iqdi_MessageSequenceNumber { ExternalAccessible := 'False'; ExternalVisible := 'False'; ExternalWritable := 'False'} : DInt;   // Message number
   END_VAR

   VAR
      s_FB_ItemError { ExternalAccessible := 'False'; ExternalVisible := 'False'; ExternalWritable := 'False'; S7_SetPoint := 'False'} : "FB_ItemError";   // Item error block's instance
      s_FB_ItemStatus { ExternalAccessible := 'False'; ExternalVisible := 'False'; ExternalWritable := 'False'; S7_SetPoint := 'False'} : "FB_ItemStatus";   // Item status block's instance
      ss_FIFOStatus { ExternalAccessible := 'False'; ExternalVisible := 'False'; ExternalWritable := 'False'; S7_SetPoint := 'False'} : "UDT_FifoStatus";   // Status structure
      s_UDT_Message { ExternalAccessible := 'False'; ExternalVisible := 'False'; ExternalWritable := 'False'; S7_SetPoint := 'False'} : "UDT_MessageV2";   // Message
      s_UDT_DimensionsCheckStatusOld { ExternalAccessible := 'False'; ExternalVisible := 'False'; ExternalWritable := 'False'; S7_SetPoint := 'False'} : "UDT_DimensionsCheckStatusV2";   // DimensionChceck  status structure
      s_UDT_ItemError { ExternalAccessible := 'False'; ExternalVisible := 'False'; ExternalWritable := 'False'; S7_SetPoint := 'False'} : "UDT_ItemError";   // Item error message body structure
      s_UDT_ItemStatus { ExternalAccessible := 'False'; ExternalVisible := 'False'; ExternalWritable := 'False'; S7_SetPoint := 'False'} : "UDT_ItemStatus";   // Item status message body structure
      s_R_TRIG_Connection {InstructionName := 'R_TRIG'; LibVersion := '1.0'; ExternalAccessible := 'False'; ExternalVisible := 'False'; ExternalWritable := 'False'; S7_SetPoint := 'False'} : R_TRIG;   // Rising edge trigger connection reastablished
      s_F_TRIG_SendAllErrors {InstructionName := 'F_TRIG'; LibVersion := '1.0'; ExternalAccessible := 'False'; ExternalVisible := 'False'; ExternalWritable := 'False'; S7_SetPoint := 'False'} : F_TRIG;   // Falling edge trigger from signal send all errors
      sdi_Code { ExternalAccessible := 'False'; ExternalVisible := 'False'; ExternalWritable := 'False'} : DInt;   // Error code
      si_ItemStatus { ExternalAccessible := 'False'; ExternalVisible := 'False'; ExternalWritable := 'False'} : Int;   // Item status
      ii_ErrorNumber { ExternalAccessible := 'False'; ExternalVisible := 'False'; ExternalWritable := 'False'} : Int;   // Counter Error Number
      si_State { ExternalAccessible := 'False'; ExternalVisible := 'False'; ExternalWritable := 'False'} : Int;   // Error state
      sx_ItemErrorMessageReq { ExternalAccessible := 'False'; ExternalVisible := 'False'; ExternalWritable := 'False'} : Bool;   // Item error message required
      sx_ItemStatusMessageReq { ExternalAccessible := 'False'; ExternalVisible := 'False'; ExternalWritable := 'False'} : Bool;   // Item status message required
      sx_SendAllProcedure { ExternalAccessible := 'False'; ExternalVisible := 'False'; ExternalWritable := 'False'} : Bool;   // Send all procedure
      sx_FIFOError { ExternalAccessible := 'False'; ExternalVisible := 'False'; ExternalWritable := 'False'} : Bool;   // FIFO error
      sx_FIFOWarning { ExternalAccessible := 'False'; ExternalVisible := 'False'; ExternalWritable := 'False'} : Bool;   // FIFO warning
      sx_ItemErrorBlockError { ExternalAccessible := 'False'; ExternalVisible := 'False'; ExternalWritable := 'False'} : Bool;   // Item error block error
      sx_ItemErrorBlockWarning { ExternalAccessible := 'False'; ExternalVisible := 'False'; ExternalWritable := 'False'} : Bool;   // Item error block warning
      sx_ItemStatusBlockError { ExternalAccessible := 'False'; ExternalVisible := 'False'; ExternalWritable := 'False'} : Bool;   // Item status block error
      sx_ItemStatusBlockWarning { ExternalAccessible := 'False'; ExternalVisible := 'False'; ExternalWritable := 'False'} : Bool;   // Item status block warning
   END_VAR


BEGIN
	(*
	----------------------------------------------------------------------------------------
	|                                                                                      |
	|  Copyright  2023             FORTNA Europe BV                                        |
	|  All Rights Reserved         Netherlands                                             |
	|                                                                                      |
	----------------------------------------------------------------------------------------
	Version history:
	Date        | Version   | Author       | Remark
	----------------------------------------------------------------------------------------
	29/03/2023  | 1.0       | M. Diebel   | Release TIA 17 | DHL Munich 2023
	13/03/2023  | 1.1       | S. Nieswiec  | Updated for new Baseline
	*)


	REGION 1 - Initialize message required signals

	    #sx_ItemErrorMessageReq := FALSE;
	    #sx_ItemStatusMessageReq := FALSE;

	    // On connection reestablish send last remembered status and error state ( status only when it's diffrent then 0 )
	    #s_R_TRIG_Connection(CLK := #ix_MFCConnected);

	    IF #s_R_TRIG_Connection.Q AND #si_ItemStatus <> 0
	    THEN
	        #sx_ItemStatusMessageReq := TRUE;
	    END_IF;

	    IF #s_R_TRIG_Connection.Q
	    THEN
	        #sx_ItemErrorMessageReq := TRUE;
	    END_IF;

	    // Prepare trigger on the collective reset signal.
	    #s_F_TRIG_SendAllErrors(CLK := #ix_SendAllErrorsState);

	    // When collective reset will go down, start send every equipment errors.
	    IF #s_F_TRIG_SendAllErrors.Q AND NOT #sx_SendAllProcedure
	    THEN
	        #ii_ErrorNumber := 0;
	        #sx_SendAllProcedure := TRUE;
	    END_IF;

	END_REGION

	REGION 2 - FIFO header status update

	    // Mode 'S' - FIFO register status update.
	    "FC_Fifo"(ic_Mode := 'S',
	              qUDT_Status => #ss_FIFOStatus,
	              qx_Error => #sx_FIFOError,
	              qx_Warning => #sx_FIFOWarning,
	              iqv_Data := #s_UDT_Message,
	              iqUDT_FifoHeader := #iq_UDT_FifoHeader,
	              iqv_DataBuffer := #iqs_FifoData);

	END_REGION

	REGION 3 - Prepare message data

	    // When there is no reset errors command, update status and errors.
	    IF NOT #ix_CollectiveReset
	        AND NOT #ss_FIFOStatus.FifoPreFull
	    THEN
	        // Status
	        IF (#i_UDT_DimensionsCheckStatus.Status <> #s_UDT_DimensionsCheckStatusOld.Status OR (#sx_SendAllProcedure AND #ii_ErrorNumber = 0))
	        THEN
	            #sx_ItemStatusMessageReq := TRUE;
	            #si_ItemStatus := #i_UDT_DimensionsCheckStatus.Status;
	            #s_UDT_DimensionsCheckStatusOld.Status := #i_UDT_DimensionsCheckStatus.Status;
	        END_IF;


